LIN {X 0,Y 374.002,Z 352.596,A -85,B 0,C 180,E1 -14322.502,E2 -14322.502} C_VEL
LIN {X 0,Y 371.832,Z 350.324,A -85,B 0,C 180,E1 -14323.336,E2 -14323.336} C_VEL
LIN {X 0,Y 368.143,Z 347.333,A -85,B 0,C 180,E1 -14324.584,E2 -14324.584} C_VEL
LIN {X 0,Y 365.076,Z 343.836,A -85,B 0,C 180,E1 -14325.586,E2 -14325.586} C_VEL
LIN {X 0,Y 361.543,Z 340.851,A -85,B 0,C 180,E1 -14326.638,E2 -14326.638} C_VEL
LIN {X 0,Y 358.551,Z 337.452,A -85,B 0,C 180,E1 -14327.482,E2 -14327.482} C_VEL
LIN {X 0,Y 355.376,Z 334.461,A -85,B 0,C 180,E1 -14328.333,E2 -14328.333} C_VEL
LIN {X 0,Y 353.051,Z 331.524,A -85,B 0,C 180,E1 -14328.94,E2 -14328.94} C_VEL
LIN {X 0,Y 350.001,Z 328.379,A -85,B 0,C 180,E1 -14329.706,E2 -14329.706} C_VEL
LIN {X 0,Y 348.216,Z 325.956,A -85,B 0,C 180,E1 -14330.137,E2 -14330.137} C_VEL
LIN {X 0,Y 345.589,Z 323.181,A -85,B 0,C 180,E1 -14330.762,E2 -14330.762} C_VEL
LIN {X 0,Y 344.015,Z 320.684,A -85,B 0,C 180,E1 -14331.145,E2 -14331.145} C_VEL
LIN {X 0,Y 341.851,Z 318.515,A -85,B 0,C 180,E1 -14331.605,E2 -14331.605} C_VEL
LIN {X 0,Y 340.82,Z 316.079,A -85,B 0,C 180,E1 -14331.984,E2 -14331.984} C_VEL
LIN {X 0,Y 340.741,Z 315.556,A -85,B 0,C 180,E1 -14332.43,E2 -14332.43} C_VEL
LIN {X 0,Y 340.767,Z 315.54,A -85,B 0,C 180,E1 -14335.664,E2 -14335.664} C_VEL
LIN {X 0,Y 340.723,Z 315.529,A -85,B 0,C 180,E1 -14338.321,E2 -14338.321} C_VEL
LIN {X 0,Y 340.692,Z 315.544,A -85,B 0,C 180,E1 -14341.044,E2 -14341.044} C_VEL
LIN {X 0,Y 340.712,Z 315.516,A -85,B 0,C 180,E1 -14345.279,E2 -14345.279} C_VEL
LIN {X 0,Y 340.708,Z 315.545,A -85,B 0,C 180,E1 -14348.387,E2 -14348.387} C_VEL
LIN {X 0,Y 340.699,Z 315.5,A -85,B 0,C 180,E1 -14352.047,E2 -14352.047} C_VEL
LIN {X 0,Y 340.714,Z 315.539,A -85,B 0,C 180,E1 -14355.468,E2 -14355.468} C_VEL
LIN {X 0,Y 340.717,Z 315.533,A -85,B 0,C 180,E1 -14358.696,E2 -14358.696} C_VEL
LIN {X 0,Y 340.731,Z 315.543,A -85,B 0,C 180,E1 -14361.773,E2 -14361.773} C_VEL
LIN {X 0,Y 340.715,Z 315.527,A -85,B 0,C 180,E1 -14365.595,E2 -14365.595} C_VEL
LIN {X 0,Y 340.716,Z 315.541,A -85,B 0,C 180,E1 -14369.571,E2 -14369.571} C_VEL
LIN {X 0,Y 340.797,Z 315.511,A -85,B 0,C 180,E1 -14373.02,E2 -14373.02} C_VEL
LIN {X 0,Y 340.753,Z 315.53,A -85,B 0,C 180,E1 -14374.697,E2 -14374.697} C_VEL
LIN {X 0,Y 340.07,Z 315.623,A -85,B 0,C 180,E1 -14375.683,E2 -14375.683} C_VEL
LIN {X 0,Y 337.176,Z 315.983,A -85,B 0,C 180,E1 -14377.288,E2 -14377.288} C_VEL
LIN {X 0,Y 334.754,Z 316.278,A -85,B 0,C 180,E1 -14378.588,E2 -14378.588} C_VEL
LIN {X 0,Y 333.755,Z 316.39,A -85,B 0,C 180,E1 -14379.595,E2 -14379.595} C_VEL
LIN {X 0,Y 333.695,Z 316.393,A -85,B 0,C 180,E1 -14379.935,E2 -14379.935} C_VEL
LIN {X 0,Y 333.738,Z 316.399,A -85,B 0,C 180,E1 -14382.854,E2 -14382.854} C_VEL
LIN {X 0,Y 333.788,Z 316.405,A -85,B 0,C 180,E1 -14386.609,E2 -14386.609} C_VEL
LIN {X 0,Y 333.842,Z 316.365,A -85,B 0,C 180,E1 -14390.305,E2 -14390.305} C_VEL
LIN {X 0,Y 333.998,Z 316.371,A -85,B 0,C 180,E1 -14392.748,E2 -14392.748} C_VEL
LIN {X 0,Y 333.802,Z 316.404,A -85,B 0,C 180,E1 -14395.17,E2 -14395.17} C_VEL
LIN {X 0,Y 334.097,Z 316.353,A -85,B 0,C 180,E1 -14397.589,E2 -14397.589} C_VEL
LIN {X 0,Y 334.22,Z 316.316,A -85,B 0,C 180,E1 -14400.001,E2 -14400.001} C_VEL
LIN {X 0,Y 334.099,Z 316.357,A -85,B 0,C 180,E1 -14402.412,E2 -14402.412} C_VEL
LIN {X 0,Y 334.007,Z 316.377,A -85,B 0,C 180,E1 -14406.04,E2 -14406.04} C_VEL
LIN {X 0,Y 333.952,Z 316.357,A -85,B 0,C 180,E1 -14408.472,E2 -14408.472} C_VEL
LIN {X 0,Y 333.784,Z 316.395,A -85,B 0,C 180,E1 -14412.156,E2 -14412.156} C_VEL
LIN {X 0,Y 333.771,Z 316.402,A -85,B 0,C 180,E1 -14415.887,E2 -14415.887} C_VEL
LIN {X 0,Y 333.79,Z 316.376,A -85,B 0,C 180,E1 -14418.655,E2 -14418.655} C_VEL
LIN {X 0,Y 333.651,Z 316.421,A -85,B 0,C 180,E1 -14422.282,E2 -14422.282} C_VEL
LIN {X 0,Y 333.729,Z 316.391,A -85,B 0,C 180,E1 -14426.247,E2 -14426.247} C_VEL
LIN {X 0,Y 333.685,Z 316.415,A -85,B 0,C 180,E1 -14428.975,E2 -14428.975} C_VEL
LIN {X 0,Y 333.639,Z 316.414,A -85,B 0,C 180,E1 -14432.588,E2 -14432.588} C_VEL
LIN {X 0,Y 333.67,Z 316.417,A -85,B 0,C 180,E1 -14436.14,E2 -14436.14} C_VEL
LIN {X 0,Y 333.643,Z 316.416,A -85,B 0,C 180,E1 -14439.194,E2 -14439.194} C_VEL
LIN {X 0,Y 333.63,Z 316.427,A -85,B 0,C 180,E1 -14442.501,E2 -14442.501} C_VEL
LIN {X 0,Y 333.594,Z 316.432,A -85,B 0,C 180,E1 -14445.956,E2 -14445.956} C_VEL
LIN {X 0,Y 333.601,Z 316.404,A -85,B 0,C 180,E1 -14449.326,E2 -14449.326} C_VEL
LIN {X 0,Y 333.662,Z 316.414,A -85,B 0,C 180,E1 -14453.169,E2 -14453.169} C_VEL
LIN {X 0,Y 333.699,Z 316.565,A -85,B 0,C 180,E1 -14456.885,E2 -14456.885} C_VEL
LIN {X 0,Y 335.008,Z 322.928,A -85,B 0,C 180,E1 -14459.332,E2 -14459.332} C_VEL
LIN {X 0,Y 336.868,Z 332.516,A -85,B 0,C 180,E1 -14462.679,E2 -14462.679} C_VEL
LIN {X 0,Y 337.066,Z 336.458,A -85,B 0,C 180,E1 -14464.033,E2 -14464.033} C_VEL
LIN {X 0,Y 336.29,Z 342.314,A -85,B 0,C 180,E1 -14465.915,E2 -14465.915} C_VEL
LIN {X 0,Y 336.975,Z 345.953,A -85,B 0,C 180,E1 -14466.117,E2 -14466.117} C_VEL
LIN {X 0,Y 342.072,Z 371.242,A -85,B 0,C 180,E1 -14467.057,E2 -14467.057} C_VEL
LIN {X 0,Y 343.729,Z 381.109,A -85,B 0,C 180,E1 -14467.391,E2 -14467.391} C_VEL
LIN {X 0,Y 342.454,Z 447.28,A -85,B 0,C 180,E1 -14468.795,E2 -14468.795} C_VEL
LIN {X 0,Y 341.879,Z 458.022,A -85,B 0,C 180,E1 -14469.152,E2 -14469.152} C_VEL
LIN {X 0,Y 341.242,Z 467.12,A -85,B 0,C 180,E1 -14469.585,E2 -14469.585} C_VEL
LIN {X 0,Y 340.44,Z 476.473,A -85,B 0,C 180,E1 -14470.164,E2 -14470.164} C_VEL
LIN {X 0,Y 339.419,Z 486.611,A -85,B 0,C 180,E1 -14470.967,E2 -14470.967} C_VEL
LIN {X 0,Y 338.379,Z 495.605,A -85,B 0,C 180,E1 -14471.848,E2 -14471.848} C_VEL
LIN {X 0,Y 337.286,Z 504.331,A -85,B 0,C 180,E1 -14472.884,E2 -14472.884} C_VEL
LIN {X 0,Y 336.298,Z 512.266,A -85,B 0,C 180,E1 -14474.013,E2 -14474.013} C_VEL
LIN {X 0,Y 335.469,Z 518.947,A -85,B 0,C 180,E1 -14475.13,E2 -14475.13} C_VEL
LIN {X 0,Y 334.69,Z 525.15,A -85,B 0,C 180,E1 -14476.336,E2 -14476.336} C_VEL
LIN {X 0,Y 333.743,Z 531.685,A -85,B 0,C 180,E1 -14477.844,E2 -14477.844} C_VEL
LIN {X 0,Y 333.24,Z 536.189,A -85,B 0,C 180,E1 -14479.059,E2 -14479.059} C_VEL
LIN {X 0,Y 332.611,Z 541.681,A -85,B 0,C 180,E1 -14480.882,E2 -14480.882} C_VEL
LIN {X 0,Y 332.203,Z 546.006,A -85,B 0,C 180,E1 -14482.708,E2 -14482.708} C_VEL
LIN {X 0,Y 332.034,Z 548.743,A -85,B 0,C 180,E1 -14484.174,E2 -14484.174} C_VEL
LIN {X 0,Y 331.97,Z 551.563,A -85,B 0,C 180,E1 -14486.359,E2 -14486.359} C_VEL
LIN {X 0,Y 331.916,Z 552.621,A -85,B 0,C 180,E1 -14487.573,E2 -14487.573} C_VEL
LIN {X 0,Y 331.913,Z 553.21,A -85,B 0,C 180,E1 -14488.787,E2 -14488.787} C_VEL
LIN {X 0,Y 331.913,Z 553.21,A -85,B 0,C 180,E1 -14491.213,E2 -14491.213} C_VEL
LIN {X 0,Y 331.916,Z 552.621,A -85,B 0,C 180,E1 -14492.427,E2 -14492.427} C_VEL
LIN {X 0,Y 331.971,Z 550.174,A -85,B 0,C 180,E1 -14494.858,E2 -14494.858} C_VEL
LIN {X 0,Y 332.106,Z 547.223,A -85,B 0,C 180,E1 -14496.684,E2 -14496.684} C_VEL
LIN {X 0,Y 332.467,Z 543.235,A -85,B 0,C 180,E1 -14498.509,E2 -14498.509} C_VEL
LIN {X 0,Y 332.988,Z 538.104,A -85,B 0,C 180,E1 -14500.335,E2 -14500.335} C_VEL
LIN {X 0,Y 333.597,Z 532.841,A -85,B 0,C 180,E1 -14501.853,E2 -14501.853} C_VEL
LIN {X 0,Y 334.485,Z 526.526,A -85,B 0,C 180,E1 -14503.363,E2 -14503.363} C_VEL
LIN {X 0,Y 335.255,Z 520.574,A -85,B 0,C 180,E1 -14504.569,E2 -14504.569} C_VEL
LIN {X 0,Y 336.287,Z 512.309,A -85,B 0,C 180,E1 -14505.981,E2 -14505.981} C_VEL
LIN {X 0,Y 337.288,Z 504.331,A -85,B 0,C 180,E1 -14507.116,E2 -14507.116} C_VEL
LIN {X 0,Y 338.395,Z 495.606,A -85,B 0,C 180,E1 -14508.151,E2 -14508.151} C_VEL
LIN {X 0,Y 339.445,Z 486.612,A -85,B 0,C 180,E1 -14509.031,E2 -14509.031} C_VEL
LIN {X 0,Y 340.43,Z 476.472,A -85,B 0,C 180,E1 -14509.836,E2 -14509.836} C_VEL
LIN {X 0,Y 341.444,Z 464.545,A -85,B 0,C 180,E1 -14510.56,E2 -14510.56} C_VEL
LIN {X 0,Y 342.275,Z 451.253,A -85,B 0,C 180,E1 -14511.098,E2 -14511.098} C_VEL
LIN {X 0,Y 342.789,Z 432.475,A -85,B 0,C 180,E1 -14511.538,E2 -14511.538} C_VEL
LIN {X 0,Y 343.621,Z 380.01,A -85,B 0,C 180,E1 -14512.641,E2 -14512.641} C_VEL
LIN {X 0,Y 338.297,Z 352.082,A -85,B 0,C 180,E1 -14513.646,E2 -14513.646} C_VEL
LIN {X 0,Y 336.284,Z 342.655,A -85,B 0,C 180,E1 -14514.04,E2 -14514.04} C_VEL
LIN {X 0,Y 336.385,Z 341.162,A -85,B 0,C 180,E1 -14514.402,E2 -14514.402} C_VEL
LIN {X 0,Y 337.123,Z 335.439,A -85,B 0,C 180,E1 -14516.307,E2 -14516.307} C_VEL
LIN {X 0,Y 336.548,Z 330.722,A -85,B 0,C 180,E1 -14517.961,E2 -14517.961} C_VEL
LIN {X 0,Y 334.829,Z 322.015,A -85,B 0,C 180,E1 -14521.09,E2 -14521.09} C_VEL
LIN {X 0,Y 333.672,Z 316.471,A -85,B 0,C 180,E1 -14523.203,E2 -14523.203} C_VEL
LIN {X 0,Y 333.662,Z 316.414,A -85,B 0,C 180,E1 -14526.831,E2 -14526.831} C_VEL
LIN {X 0,Y 333.602,Z 316.404,A -85,B 0,C 180,E1 -14530.773,E2 -14530.773} C_VEL
LIN {X 0,Y 333.591,Z 316.43,A -85,B 0,C 180,E1 -14534.249,E2 -14534.249} C_VEL
LIN {X 0,Y 333.639,Z 316.427,A -85,B 0,C 180,E1 -14537.617,E2 -14537.617} C_VEL
LIN {X 0,Y 333.649,Z 316.416,A -85,B 0,C 180,E1 -14541.201,E2 -14541.201} C_VEL
LIN {X 0,Y 333.67,Z 316.417,A -85,B 0,C 180,E1 -14543.86,E2 -14543.86} C_VEL
LIN {X 0,Y 333.639,Z 316.414,A -85,B 0,C 180,E1 -14547.412,E2 -14547.412} C_VEL
LIN {X 0,Y 333.685,Z 316.415,A -85,B 0,C 180,E1 -14551.025,E2 -14551.025} C_VEL
LIN {X 0,Y 333.729,Z 316.391,A -85,B 0,C 180,E1 -14553.753,E2 -14553.753} C_VEL
LIN {X 0,Y 333.651,Z 316.421,A -85,B 0,C 180,E1 -14557.718,E2 -14557.718} C_VEL
LIN {X 0,Y 333.787,Z 316.377,A -85,B 0,C 180,E1 -14561.588,E2 -14561.588} C_VEL
LIN {X 0,Y 333.802,Z 316.405,A -85,B 0,C 180,E1 -14565.576,E2 -14565.576} C_VEL
LIN {X 0,Y 333.827,Z 316.377,A -85,B 0,C 180,E1 -14569.077,E2 -14569.077} C_VEL
LIN {X 0,Y 333.999,Z 316.366,A -85,B 0,C 180,E1 -14572.746,E2 -14572.746} C_VEL
LIN {X 0,Y 333.802,Z 316.406,A -85,B 0,C 180,E1 -14575.168,E2 -14575.168} C_VEL
LIN {X 0,Y 334.099,Z 316.357,A -85,B 0,C 180,E1 -14577.588,E2 -14577.588} C_VEL
LIN {X 0,Y 334.22,Z 316.316,A -85,B 0,C 180,E1 -14579.999,E2 -14579.999} C_VEL
LIN {X 0,Y 334.097,Z 316.353,A -85,B 0,C 180,E1 -14582.411,E2 -14582.411} C_VEL
LIN {X 0,Y 333.983,Z 316.373,A -85,B 0,C 180,E1 -14586.674,E2 -14586.674} C_VEL
LIN {X 0,Y 333.842,Z 316.365,A -85,B 0,C 180,E1 -14589.695,E2 -14589.695} C_VEL
LIN {X 0,Y 333.788,Z 316.405,A -85,B 0,C 180,E1 -14593.391,E2 -14593.391} C_VEL
LIN {X 0,Y 333.738,Z 316.399,A -85,B 0,C 180,E1 -14597.146,E2 -14597.146} C_VEL
LIN {X 0,Y 333.729,Z 316.388,A -85,B 0,C 180,E1 -14599.69,E2 -14599.69} C_VEL
LIN {X 0,Y 333.684,Z 316.415,A -85,B 0,C 180,E1 -14602.278,E2 -14602.278} C_VEL
LIN {X 0,Y 333.728,Z 316.398,A -85,B 0,C 180,E1 -14606.246,E2 -14606.246} C_VEL
LIN {X 0,Y 333.703,Z 316.404,A -85,B 0,C 180,E1 -14608.972,E2 -14608.972} C_VEL
LIN {X 0,Y 333.638,Z 316.421,A -85,B 0,C 180,E1 -14612.588,E2 -14612.588} C_VEL
LIN {X 0,Y 333.669,Z 316.414,A -85,B 0,C 180,E1 -14616.139,E2 -14616.139} C_VEL
LIN {X 0,Y 333.677,Z 316.415,A -85,B 0,C 180,E1 -14619.187,E2 -14619.187} C_VEL
LIN {X 0,Y 333.681,Z 316.417,A -85,B 0,C 180,E1 -14622.511,E2 -14622.511} C_VEL
LIN {X 0,Y 333.628,Z 316.401,A -85,B 0,C 180,E1 -14625.962,E2 -14625.962} C_VEL
LIN {X 0,Y 333.648,Z 316.388,A -85,B 0,C 180,E1 -14629.314,E2 -14629.314} C_VEL
LIN {X 0,Y 333.649,Z 316.427,A -85,B 0,C 180,E1 -14632.35,E2 -14632.35} C_VEL
LIN {X 0,Y 333.668,Z 316.39,A -85,B 0,C 180,E1 -14635.342,E2 -14635.342} C_VEL
LIN {X 0,Y 333.684,Z 316.406,A -85,B 0,C 180,E1 -14639.637,E2 -14639.637} C_VEL
LIN {X 0,Y 333.734,Z 316.411,A -85,B 0,C 180,E1 -14642.401,E2 -14642.401} C_VEL
LIN {X 0,Y 333.722,Z 316.418,A -85,B 0,C 180,E1 -14645.091,E2 -14645.091} C_VEL
LIN {X 0,Y 333.713,Z 316.564,A -85,B 0,C 180,E1 -14646.636,E2 -14646.636} C_VEL
LIN {X 0,Y 333.901,Z 317.484,A -85,B 0,C 180,E1 -14646.906,E2 -14646.906} C_VEL
LIN {X 0,Y 335.44,Z 320.272,A -85,B 0,C 180,E1 -14647.294,E2 -14647.294} C_VEL
LIN {X 0,Y 337.24,Z 322.145,A -85,B 0,C 180,E1 -14647.649,E2 -14647.649} C_VEL
LIN {X 0,Y 339.606,Z 325.545,A -85,B 0,C 180,E1 -14648.193,E2 -14648.193} C_VEL
LIN {X 0,Y 341.243,Z 327.304,A -85,B 0,C 180,E1 -14648.55,E2 -14648.55} C_VEL
LIN {X 0,Y 344.017,Z 330.834,A -85,B 0,C 180,E1 -14649.167,E2 -14649.167} C_VEL
LIN {X 0,Y 346.131,Z 333.088,A -85,B 0,C 180,E1 -14649.669,E2 -14649.669} C_VEL
LIN {X 0,Y 349.257,Z 336.713,A -85,B 0,C 180,E1 -14650.409,E2 -14650.409} C_VEL
LIN {X 0,Y 351.305,Z 338.801,A -85,B 0,C 180,E1 -14650.915,E2 -14650.915} C_VEL
LIN {X 0,Y 354.984,Z 342.849,A -85,B 0,C 180,E1 -14651.859,E2 -14651.859} C_VEL
LIN {X 0,Y 357.12,Z 344.835,A -85,B 0,C 180,E1 -14652.431,E2 -14652.431} C_VEL
LIN {X 0,Y 360.924,Z 348.801,A -85,B 0,C 180,E1 -14653.498,E2 -14653.498} C_VEL
LIN {X 0,Y 363.731,Z 351.163,A -85,B 0,C 180,E1 -14654.333,E2 -14654.333} C_VEL
LIN {X 0,Y 367.168,Z 354.797,A -85,B 0,C 180,E1 -14655.432,E2 -14655.432} C_VEL
LIN {X 0,Y 371.068,Z 357.902,A -85,B 0,C 180,E1 -14656.751,E2 -14656.751} C_VEL
LIN {X 0,Y 374.707,Z 361.571,A -85,B 0,C 180,E1 -14658.165,E2 -14658.165} C_VEL
LIN {X 0,Y 378.245,Z 364.068,A -85,B 0,C 180,E1 -14659.673,E2 -14659.673} C_VEL
LIN {X 0,Y 379.884,Z 365.154,A -85,B 0,C 180,E1 -14660.464,E2 -14660.464} C_VEL
LIN {X 0,Y 382.521,Z 368.124,A -85,B 0,C 180,E1 -14661.961,E2 -14661.961} C_VEL
LIN {X 0,Y 384.968,Z 370.062,A -85,B 0,C 180,E1 -14663.58,E2 -14663.58} C_VEL
LIN {X 0,Y 387.283,Z 371.337,A -85,B 0,C 180,E1 -14665.578,E2 -14665.578} C_VEL
LIN {X 0,Y 388.664,Z 371.823,A -85,B 0,C 180,E1 -14667.428,E2 -14667.428} C_VEL
LIN {X 0,Y 389.239,Z 372.261,A -85,B 0,C 180,E1 -14668.965,E2 -14668.965} C_VEL
LIN {X 0,Y 389.407,Z 372.18,A -85,B 0,C 180,E1 -14670,E2 -14670} C_VEL
LIN {X 0,Y 389.126,Z 372.136,A -85,B 0,C 180,E1 -14671.552,E2 -14671.552} C_VEL
LIN {X 0,Y 388.36,Z 371.702,A -85,B 0,C 180,E1 -14673.112,E2 -14673.112} C_VEL
LIN {X 0,Y 386.736,Z 371.099,A -85,B 0,C 180,E1 -14674.943,E2 -14674.943} C_VEL
LIN {X 0,Y 384.56,Z 369.785,A -85,B 0,C 180,E1 -14676.7,E2 -14676.7} C_VEL
LIN {X 0,Y 382.058,Z 367.692,A -85,B 0,C 180,E1 -14678.309,E2 -14678.309} C_VEL
LIN {X 0,Y 379.212,Z 364.566,A -85,B 0,C 180,E1 -14679.865,E2 -14679.865} C_VEL
LIN {X 0,Y 375.944,Z 362.622,A -85,B 0,C 180,E1 -14681.307,E2 -14681.307} C_VEL
LIN {X 0,Y 372.666,Z 359.673,A -85,B 0,C 180,E1 -14682.629,E2 -14682.629} C_VEL
LIN {X 0,Y 370.003,Z 356.954,A -85,B 0,C 180,E1 -14683.635,E2 -14683.635} C_VEL
LIN {X 0,Y 365.937,Z 353.626,A -85,B 0,C 180,E1 -14684.976,E2 -14684.976} C_VEL
LIN {X 0,Y 362.653,Z 350.169,A -85,B 0,C 180,E1 -14685.995,E2 -14685.995} C_VEL
LIN {X 0,Y 358.82,Z 346.809,A -85,B 0,C 180,E1 -14687.085,E2 -14687.085} C_VEL
LIN {X 0,Y 355.812,Z 343.521,A -85,B 0,C 180,E1 -14687.928,E2 -14687.928} C_VEL
LIN {X 0,Y 352.062,Z 339.815,A -85,B 0,C 180,E1 -14688.881,E2 -14688.881} C_VEL
LIN {X 0,Y 350.013,Z 337.385,A -85,B 0,C 180,E1 -14689.415,E2 -14689.415} C_VEL
LIN {X 0,Y 346.537,Z 333.696,A -85,B 0,C 180,E1 -14690.229,E2 -14690.229} C_VEL
LIN {X 0,Y 344.964,Z 331.748,A -85,B 0,C 180,E1 -14690.614,E2 -14690.614} C_VEL
LIN {X 0,Y 341.952,Z 328.424,A -85,B 0,C 180,E1 -14691.286,E2 -14691.286} C_VEL
LIN {X 0,Y 340.285,Z 326.164,A -85,B 0,C 180,E1 -14691.661,E2 -14691.661} C_VEL
LIN {X 0,Y 337.899,Z 323.317,A -85,B 0,C 180,E1 -14692.197,E2 -14692.197} C_VEL
LIN {X 0,Y 336.543,Z 321.282,A -85,B 0,C 180,E1 -14692.493,E2 -14692.493} C_VEL
LIN {X 0,Y 334.616,Z 319.146,A -85,B 0,C 180,E1 -14692.878,E2 -14692.878} C_VEL
LIN {X 0,Y 333.801,Z 317.073,A -85,B 0,C 180,E1 -14693.17,E2 -14693.17} C_VEL
LIN {X 0,Y 333.679,Z 316.494,A -85,B 0,C 180,E1 -14693.425,E2 -14693.425} C_VEL
LIN {X 0,Y 333.73,Z 316.416,A -85,B 0,C 180,E1 -14696.246,E2 -14696.246} C_VEL
LIN {X 0,Y 333.684,Z 316.4,A -85,B 0,C 180,E1 -14698.974,E2 -14698.974} C_VEL
LIN {X 0,Y 333.637,Z 316.42,A -85,B 0,C 180,E1 -14702.587,E2 -14702.587} C_VEL
LIN {X 0,Y 333.671,Z 316.404,A -85,B 0,C 180,E1 -14706.139,E2 -14706.139} C_VEL
LIN {X 0,Y 333.664,Z 316.414,A -85,B 0,C 180,E1 -14709.189,E2 -14709.189} C_VEL
LIN {X 0,Y 333.631,Z 316.38,A -85,B 0,C 180,E1 -14712.501,E2 -14712.501} C_VEL
LIN {X 0,Y 333.661,Z 316.423,A -85,B 0,C 180,E1 -14715.967,E2 -14715.967} C_VEL
LIN {X 0,Y 333.694,Z 316.405,A -85,B 0,C 180,E1 -14719.304,E2 -14719.304} C_VEL
LIN {X 0,Y 333.658,Z 316.422,A -85,B 0,C 180,E1 -14723.168,E2 -14723.168} C_VEL
LIN {X 0,Y 333.631,Z 316.415,A -85,B 0,C 180,E1 -14726.792,E2 -14726.792} C_VEL
LIN {X 0,Y 333.695,Z 316.416,A -85,B 0,C 180,E1 -14729.71,E2 -14729.71} C_VEL
LIN {X 0,Y 333.736,Z 316.39,A -85,B 0,C 180,E1 -14732.401,E2 -14732.401} C_VEL
LIN {X 0,Y 333.718,Z 316.41,A -85,B 0,C 180,E1 -14735.091,E2 -14735.091} C_VEL
LIN {X 0,Y 333.672,Z 316.406,A -85,B 0,C 180,E1 -14739.019,E2 -14739.019} C_VEL
LIN {X 0,Y 333.695,Z 316.393,A -85,B 0,C 180,E1 -14739.935,E2 -14739.935} C_VEL
LIN {X 0,Y 333.085,Z 316.469,A -85,B 0,C 180,E1 -14740.943,E2 -14740.943} C_VEL
LIN {X 0,Y 330.261,Z 316.836,A -85,B 0,C 180,E1 -14742.582,E2 -14742.582} C_VEL
LIN {X 0,Y 327.845,Z 317.148,A -85,B 0,C 180,E1 -14743.91,E2 -14743.91} C_VEL
LIN {X 0,Y 326.823,Z 317.277,A -85,B 0,C 180,E1 -14744.938,E2 -14744.938} C_VEL
LIN {X 0,Y 326.75,Z 317.284,A -85,B 0,C 180,E1 -14745.286,E2 -14745.286} C_VEL
LIN {X 0,Y 326.761,Z 317.253,A -85,B 0,C 180,E1 -14748.839,E2 -14748.839} C_VEL
LIN {X 0,Y 326.95,Z 317.247,A -85,B 0,C 180,E1 -14752.59,E2 -14752.59} C_VEL
LIN {X 0,Y 326.768,Z 317.281,A -85,B 0,C 180,E1 -14755.065,E2 -14755.065} C_VEL
LIN {X 0,Y 327.038,Z 317.232,A -85,B 0,C 180,E1 -14757.537,E2 -14757.537} C_VEL
LIN {X 0,Y 327.172,Z 317.193,A -85,B 0,C 180,E1 -14760.001,E2 -14760.001} C_VEL
LIN {X 0,Y 327.04,Z 317.236,A -85,B 0,C 180,E1 -14762.464,E2 -14762.464} C_VEL
LIN {X 0,Y 326.982,Z 317.252,A -85,B 0,C 180,E1 -14766.17,E2 -14766.17} C_VEL
LIN {X 0,Y 326.799,Z 317.241,A -85,B 0,C 180,E1 -14769.907,E2 -14769.907} C_VEL
LIN {X 0,Y 326.753,Z 317.279,A -85,B 0,C 180,E1 -14773.686,E2 -14773.686} C_VEL
LIN {X 0,Y 326.693,Z 317.266,A -85,B 0,C 180,E1 -14777.529,E2 -14777.529} C_VEL
LIN {X 0,Y 326.652,Z 317.275,A -85,B 0,C 180,E1 -14780.136,E2 -14780.136} C_VEL
LIN {X 0,Y 326.643,Z 317.293,A -85,B 0,C 180,E1 -14784.13,E2 -14784.13} C_VEL
LIN {X 0,Y 326.678,Z 317.267,A -85,B 0,C 180,E1 -14786.859,E2 -14786.859} C_VEL
LIN {X 0,Y 326.63,Z 317.299,A -85,B 0,C 180,E1 -14790.611,E2 -14790.611} C_VEL
LIN {X 0,Y 326.602,Z 317.282,A -85,B 0,C 180,E1 -14794.021,E2 -14794.021} C_VEL
LIN {X 0,Y 326.623,Z 317.298,A -85,B 0,C 180,E1 -14797.239,E2 -14797.239} C_VEL
LIN {X 0,Y 326.575,Z 317.301,A -85,B 0,C 180,E1 -14801.132,E2 -14801.132} C_VEL
LIN {X 0,Y 326.525,Z 317.305,A -85,B 0,C 180,E1 -14804.744,E2 -14804.744} C_VEL
LIN {X 0,Y 326.561,Z 317.29,A -85,B 0,C 180,E1 -14808.153,E2 -14808.153} C_VEL
LIN {X 0,Y 326.581,Z 317.301,A -85,B 0,C 180,E1 -14811.387,E2 -14811.387} C_VEL
LIN {X 0,Y 326.618,Z 317.286,A -85,B 0,C 180,E1 -14814.853,E2 -14814.853} C_VEL
LIN {X 0,Y 326.672,Z 317.479,A -85,B 0,C 180,E1 -14816.487,E2 -14816.487} C_VEL
LIN {X 0,Y 328.006,Z 324.056,A -85,B 0,C 180,E1 -14819.055,E2 -14819.055} C_VEL
LIN {X 0,Y 329.631,Z 332.307,A -85,B 0,C 180,E1 -14822.028,E2 -14822.028} C_VEL
LIN {X 0,Y 330.177,Z 336.26,A -85,B 0,C 180,E1 -14823.45,E2 -14823.45} C_VEL
LIN {X 0,Y 329.446,Z 342.132,A -85,B 0,C 180,E1 -14825.385,E2 -14825.385} C_VEL
LIN {X 0,Y 330.305,Z 346.413,A -85,B 0,C 180,E1 -14825.619,E2 -14825.619} C_VEL
LIN {X 0,Y 335.111,Z 370.101,A -85,B 0,C 180,E1 -14826.53,E2 -14826.53} C_VEL
LIN {X 0,Y 337.185,Z 382.571,A -85,B 0,C 180,E1 -14826.965,E2 -14826.965} C_VEL
LIN {X 0,Y 335.845,Z 447.093,A -85,B 0,C 180,E1 -14828.357,E2 -14828.357} C_VEL
LIN {X 0,Y 335.267,Z 457.829,A -85,B 0,C 180,E1 -14828.721,E2 -14828.721} C_VEL
LIN {X 0,Y 334.61,Z 466.926,A -85,B 0,C 180,E1 -14829.161,E2 -14829.161} C_VEL
LIN {X 0,Y 333.75,Z 476.278,A -85,B 0,C 180,E1 -14829.749,E2 -14829.749} C_VEL
LIN {X 0,Y 332.695,Z 486.417,A -85,B 0,C 180,E1 -14830.567,E2 -14830.567} C_VEL
LIN {X 0,Y 331.616,Z 495.411,A -85,B 0,C 180,E1 -14831.465,E2 -14831.465} C_VEL
LIN {X 0,Y 330.49,Z 504.137,A -85,B 0,C 180,E1 -14832.52,E2 -14832.52} C_VEL
LIN {X 0,Y 329.478,Z 511.897,A -85,B 0,C 180,E1 -14833.644,E2 -14833.644} C_VEL
LIN {X 0,Y 328.582,Z 518.809,A -85,B 0,C 180,E1 -14834.822,E2 -14834.822} C_VEL
LIN {X 0,Y 327.778,Z 524.956,A -85,B 0,C 180,E1 -14836.042,E2 -14836.042} C_VEL
LIN {X 0,Y 326.779,Z 531.49,A -85,B 0,C 180,E1 -14837.581,E2 -14837.581} C_VEL
LIN {X 0,Y 326.216,Z 535.993,A -85,B 0,C 180,E1 -14838.82,E2 -14838.82} C_VEL
LIN {X 0,Y 325.578,Z 541.486,A -85,B 0,C 180,E1 -14840.683,E2 -14840.683} C_VEL
LIN {X 0,Y 325.154,Z 545.812,A -85,B 0,C 180,E1 -14842.549,E2 -14842.549} C_VEL
LIN {X 0,Y 324.926,Z 548.844,A -85,B 0,C 180,E1 -14844.251,E2 -14844.251} C_VEL
LIN {X 0,Y 324.877,Z 551.369,A -85,B 0,C 180,E1 -14846.279,E2 -14846.279} C_VEL
LIN {X 0,Y 324.835,Z 552.427,A -85,B 0,C 180,E1 -14847.52,E2 -14847.52} C_VEL
LIN {X 0,Y 324.822,Z 553.016,A -85,B 0,C 180,E1 -14848.76,E2 -14848.76} C_VEL
LIN {X 0,Y 324.822,Z 553.016,A -85,B 0,C 180,E1 -14851.24,E2 -14851.24} C_VEL
LIN {X 0,Y 324.835,Z 552.427,A -85,B 0,C 180,E1 -14852.48,E2 -14852.48} C_VEL
LIN {X 0,Y 324.882,Z 549.979,A -85,B 0,C 180,E1 -14854.964,E2 -14854.964} C_VEL
LIN {X 0,Y 325.047,Z 547.029,A -85,B 0,C 180,E1 -14856.83,E2 -14856.83} C_VEL
LIN {X 0,Y 325.406,Z 543.04,A -85,B 0,C 180,E1 -14858.695,E2 -14858.695} C_VEL
LIN {X 0,Y 325.968,Z 537.909,A -85,B 0,C 180,E1 -14860.56,E2 -14860.56} C_VEL
LIN {X 0,Y 326.628,Z 532.646,A -85,B 0,C 180,E1 -14862.11,E2 -14862.11} C_VEL
LIN {X 0,Y 327.57,Z 526.331,A -85,B 0,C 180,E1 -14863.651,E2 -14863.651} C_VEL
LIN {X 0,Y 328.346,Z 520.379,A -85,B 0,C 180,E1 -14864.883,E2 -14864.883} C_VEL
LIN {X 0,Y 329.338,Z 512.888,A -85,B 0,C 180,E1 -14866.199,E2 -14866.199} C_VEL
LIN {X 0,Y 330.332,Z 505.271,A -85,B 0,C 180,E1 -14867.329,E2 -14867.329} C_VEL
LIN {X 0,Y 331.498,Z 496.764,A -85,B 0,C 180,E1 -14868.382,E2 -14868.382} C_VEL
LIN {X 0,Y 332.563,Z 488.05,A -85,B 0,C 180,E1 -14869.28,E2 -14869.28} C_VEL
LIN {X 0,Y 333.576,Z 478.293,A -85,B 0,C 180,E1 -14870.101,E2 -14870.101} C_VEL
LIN {X 0,Y 334.398,Z 469.501,A -85,B 0,C 180,E1 -14870.692,E2 -14870.692} C_VEL
LIN {X 0,Y 335.115,Z 459.576,A -85,B 0,C 180,E1 -14871.208,E2 -14871.208} C_VEL
LIN {X 0,Y 335.735,Z 449.728,A -85,B 0,C 180,E1 -14871.57,E2 -14871.57} C_VEL
LIN {X 0,Y 336.287,Z 428.702,A -85,B 0,C 180,E1 -14872.056,E2 -14872.056} C_VEL
LIN {X 0,Y 337.081,Z 381.176,A -85,B 0,C 180,E1 -14873.075,E2 -14873.075} C_VEL
LIN {X 0,Y 332.125,Z 354.829,A -85,B 0,C 180,E1 -14874.045,E2 -14874.045} C_VEL
LIN {X 0,Y 329.474,Z 342.433,A -85,B 0,C 180,E1 -14874.572,E2 -14874.572} C_VEL
LIN {X 0,Y 329.57,Z 340.965,A -85,B 0,C 180,E1 -14874.941,E2 -14874.941} C_VEL
LIN {X 0,Y 330.155,Z 336.089,A -85,B 0,C 180,E1 -14876.612,E2 -14876.612} C_VEL
LIN {X 0,Y 329.18,Z 329.742,A -85,B 0,C 180,E1 -14878.912,E2 -14878.912} C_VEL
LIN {X 0,Y 327.232,Z 320.188,A -85,B 0,C 180,E1 -14882.474,E2 -14882.474} C_VEL
LIN {X 0,Y 326.639,Z 317.378,A -85,B 0,C 180,E1 -14883.587,E2 -14883.587} C_VEL
LIN {X 0,Y 326.622,Z 317.296,A -85,B 0,C 180,E1 -14887.236,E2 -14887.236} C_VEL
LIN {X 0,Y 326.542,Z 317.285,A -85,B 0,C 180,E1 -14891.123,E2 -14891.123} C_VEL
LIN {X 0,Y 326.559,Z 317.309,A -85,B 0,C 180,E1 -14893.525,E2 -14893.525} C_VEL
LIN {X 0,Y 326.574,Z 317.303,A -85,B 0,C 180,E1 -14897.027,E2 -14897.027} C_VEL
LIN {X 0,Y 326.608,Z 317.292,A -85,B 0,C 180,E1 -14900.772,E2 -14900.772} C_VEL
LIN {X 0,Y 326.607,Z 317.292,A -85,B 0,C 180,E1 -14904.479,E2 -14904.479} C_VEL
LIN {X 0,Y 326.604,Z 317.29,A -85,B 0,C 180,E1 -14907.454,E2 -14907.454} C_VEL
LIN {X 0,Y 326.643,Z 317.293,A -85,B 0,C 180,E1 -14910.339,E2 -14910.339} C_VEL
LIN {X 0,Y 326.685,Z 317.276,A -85,B 0,C 180,E1 -14914.515,E2 -14914.515} C_VEL
LIN {X 0,Y 326.614,Z 317.294,A -85,B 0,C 180,E1 -14918.542,E2 -14918.542} C_VEL
LIN {X 0,Y 326.739,Z 317.254,A -85,B 0,C 180,E1 -14921.177,E2 -14921.177} C_VEL
LIN {X 0,Y 326.757,Z 317.281,A -85,B 0,C 180,E1 -14925.432,E2 -14925.432} C_VEL
LIN {X 0,Y 326.763,Z 317.26,A -85,B 0,C 180,E1 -14928.838,E2 -14928.838} C_VEL
LIN {X 0,Y 326.951,Z 317.243,A -85,B 0,C 180,E1 -14932.589,E2 -14932.589} C_VEL
LIN {X 0,Y 326.769,Z 317.281,A -85,B 0,C 180,E1 -14935.064,E2 -14935.064} C_VEL
LIN {X 0,Y 327.04,Z 317.236,A -85,B 0,C 180,E1 -14937.536,E2 -14937.536} C_VEL
LIN {X 0,Y 327.172,Z 317.193,A -85,B 0,C 180,E1 -14939.999,E2 -14939.999} C_VEL
LIN {X 0,Y 327.038,Z 317.232,A -85,B 0,C 180,E1 -14942.463,E2 -14942.463} C_VEL
LIN {X 0,Y 326.95,Z 317.25,A -85,B 0,C 180,E1 -14946.666,E2 -14946.666} C_VEL
LIN {X 0,Y 326.797,Z 317.241,A -85,B 0,C 180,E1 -14949.906,E2 -14949.906} C_VEL
LIN {X 0,Y 326.751,Z 317.282,A -85,B 0,C 180,E1 -14953.685,E2 -14953.685} C_VEL
LIN {X 0,Y 326.691,Z 317.273,A -85,B 0,C 180,E1 -14957.528,E2 -14957.528} C_VEL
LIN {X 0,Y 326.655,Z 317.272,A -85,B 0,C 180,E1 -14960.135,E2 -14960.135} C_VEL
LIN {X 0,Y 326.644,Z 317.295,A -85,B 0,C 180,E1 -14964.129,E2 -14964.129} C_VEL
LIN {X 0,Y 326.677,Z 317.27,A -85,B 0,C 180,E1 -14966.857,E2 -14966.857} C_VEL
LIN {X 0,Y 326.631,Z 317.298,A -85,B 0,C 180,E1 -14970.611,E2 -14970.611} C_VEL
LIN {X 0,Y 326.6,Z 317.286,A -85,B 0,C 180,E1 -14974.019,E2 -14974.019} C_VEL
LIN {X 0,Y 326.622,Z 317.301,A -85,B 0,C 180,E1 -14977.239,E2 -14977.239} C_VEL
LIN {X 0,Y 326.628,Z 317.286,A -85,B 0,C 180,E1 -14980.203,E2 -14980.203} C_VEL
LIN {X 0,Y 326.611,Z 317.3,A -85,B 0,C 180,E1 -14983.516,E2 -14983.516} C_VEL
LIN {X 0,Y 326.582,Z 317.261,A -85,B 0,C 180,E1 -14987.026,E2 -14987.026} C_VEL
LIN {X 0,Y 326.626,Z 317.29,A -85,B 0,C 180,E1 -14990.768,E2 -14990.768} C_VEL
LIN {X 0,Y 326.607,Z 317.274,A -85,B 0,C 180,E1 -14994.481,E2 -14994.481} C_VEL
LIN {X 0,Y 326.602,Z 317.296,A -85,B 0,C 180,E1 -14997.456,E2 -14997.456} C_VEL
LIN {X 0,Y 326.642,Z 317.277,A -85,B 0,C 180,E1 -15000.34,E2 -15000.34} C_VEL
LIN {X 0,Y 326.685,Z 317.294,A -85,B 0,C 180,E1 -15004.516,E2 -15004.516} C_VEL
LIN {X 0,Y 326.69,Z 317.588,A -85,B 0,C 180,E1 -15005.621,E2 -15005.621} C_VEL
LIN {X 0,Y 327.047,Z 318.932,A -85,B 0,C 180,E1 -15005.866,E2 -15005.866} C_VEL
LIN {X 0,Y 328.752,Z 321.563,A -85,B 0,C 180,E1 -15006.21,E2 -15006.21} C_VEL
LIN {X 0,Y 329.922,Z 322.861,A -85,B 0,C 180,E1 -15006.429,E2 -15006.429} C_VEL
LIN {X 0,Y 332.332,Z 326.359,A -85,B 0,C 180,E1 -15006.946,E2 -15006.946} C_VEL
LIN {X 0,Y 333.847,Z 328.148,A -85,B 0,C 180,E1 -15007.255,E2 -15007.255} C_VEL
LIN {X 0,Y 336.858,Z 331.835,A -85,B 0,C 180,E1 -15007.874,E2 -15007.874} C_VEL
LIN {X 0,Y 341.329,Z 337.18,A -85,B 0,C 180,E1 -15008.865,E2 -15008.865} C_VEL
LIN {X 0,Y 343.577,Z 339.682,A -85,B 0,C 180,E1 -15009.36,E2 -15009.36} C_VEL
LIN {X 0,Y 347.348,Z 343.653,A -85,B 0,C 180,E1 -15010.249,E2 -15010.249} C_VEL
LIN {X 0,Y 352.042,Z 348.766,A -85,B 0,C 180,E1 -15011.415,E2 -15011.415} C_VEL
LIN {X 0,Y 354.731,Z 351.21,A -85,B 0,C 180,E1 -15012.089,E2 -15012.089} C_VEL
LIN {X 0,Y 358.929,Z 355.424,A -85,B 0,C 180,E1 -15013.243,E2 -15013.243} C_VEL
LIN {X 0,Y 361.622,Z 357.669,A -85,B 0,C 180,E1 -15014.013,E2 -15014.013} C_VEL
LIN {X 0,Y 365.635,Z 361.687,A -85,B 0,C 180,E1 -15015.258,E2 -15015.258} C_VEL
LIN {X 0,Y 369.617,Z 364.847,A -85,B 0,C 180,E1 -15016.584,E2 -15016.584} C_VEL
LIN {X 0,Y 373.295,Z 368.422,A -85,B 0,C 180,E1 -15017.979,E2 -15017.979} C_VEL
LIN {X 0,Y 377.095,Z 371.047,A -85,B 0,C 180,E1 -15019.567,E2 -15019.567} C_VEL
LIN {X 0,Y 378.503,Z 371.984,A -85,B 0,C 180,E1 -15020.245,E2 -15020.245} C_VEL
LIN {X 0,Y 381.112,Z 374.829,A -85,B 0,C 180,E1 -15021.67,E2 -15021.67} C_VEL
LIN {X 0,Y 383.334,Z 376.638,A -85,B 0,C 180,E1 -15023.062,E2 -15023.062} C_VEL
LIN {X 0,Y 385.526,Z 377.999,A -85,B 0,C 180,E1 -15024.77,E2 -15024.77} C_VEL
LIN {X 0,Y 387.235,Z 378.642,A -85,B 0,C 180,E1 -15026.554,E2 -15026.554} C_VEL
LIN {X 0,Y 388.257,Z 379.202,A -85,B 0,C 180,E1 -15028.444,E2 -15028.444} C_VEL
LIN {X 0,Y 388.542,Z 379.227,A -85,B 0,C 180,E1 -15030,E2 -15030} C_VEL
LIN {X 0,Y 388.257,Z 379.184,A -85,B 0,C 180,E1 -15031.556,E2 -15031.556} C_VEL
LIN {X 0,Y 387.234,Z 378.67,A -85,B 0,C 180,E1 -15033.443,E2 -15033.443} C_VEL
LIN {X 0,Y 385.526,Z 378,A -85,B 0,C 180,E1 -15035.23,E2 -15035.23} C_VEL
LIN {X 0,Y 383.278,Z 376.595,A -85,B 0,C 180,E1 -15036.977,E2 -15036.977} C_VEL
LIN {X 0,Y 380.599,Z 374.308,A -85,B 0,C 180,E1 -15038.639,E2 -15038.639} C_VEL
LIN {X 0,Y 377.707,Z 371.348,A -85,B 0,C 180,E1 -15040.146,E2 -15040.146} C_VEL
LIN {X 0,Y 373.851,Z 368.917,A -85,B 0,C 180,E1 -15041.791,E2 -15041.791} C_VEL
LIN {X 0,Y 369.775,Z 365.065,A -85,B 0,C 180,E1 -15043.355,E2 -15043.355} C_VEL
LIN {X 0,Y 367.883,Z 363.434,A -85,B 0,C 180,E1 -15043.999,E2 -15043.999} C_VEL
LIN {X 0,Y 363.711,Z 359.953,A -85,B 0,C 180,E1 -15045.341,E2 -15045.341} C_VEL
LIN {X 0,Y 360.454,Z 356.588,A -85,B 0,C 180,E1 -15046.335,E2 -15046.335} C_VEL
LIN {X 0,Y 356.027,Z 352.677,A -85,B 0,C 180,E1 -15047.557,E2 -15047.557} C_VEL
LIN {X 0,Y 353.026,Z 349.612,A -85,B 0,C 180,E1 -15048.342,E2 -15048.342} C_VEL
LIN {X 0,Y 349.006,Z 345.521,A -85,B 0,C 180,E1 -15049.361,E2 -15049.361} C_VEL
LIN {X 0,Y 346.947,Z 343.303,A -85,B 0,C 180,E1 -15049.842,E2 -15049.842} C_VEL
LIN {X 0,Y 343.168,Z 339.146,A -85,B 0,C 180,E1 -15050.737,E2 -15050.737} C_VEL
LIN {X 0,Y 338.397,Z 333.83,A -85,B 0,C 180,E1 -15051.778,E2 -15051.778} C_VEL
LIN {X 0,Y 336.613,Z 331.601,A -85,B 0,C 180,E1 -15052.177,E2 -15052.177} C_VEL
LIN {X 0,Y 333.567,Z 327.726,A -85,B 0,C 180,E1 -15052.804,E2 -15052.804} C_VEL
LIN {X 0,Y 330.473,Z 323.86,A -85,B 0,C 180,E1 -15053.449,E2 -15053.449} C_VEL
LIN {X 0,Y 329.168,Z 321.932,A -85,B 0,C 180,E1 -15053.716,E2 -15053.716} C_VEL
LIN {X 0,Y 327.279,Z 319.491,A -85,B 0,C 180,E1 -15054.079,E2 -15054.079} C_VEL
LIN {X 0,Y 326.716,Z 317.711,A -85,B 0,C 180,E1 -15054.334,E2 -15054.334} C_VEL
LIN {X 0,Y 326.683,Z 317.294,A -85,B 0,C 180,E1 -15054.803,E2 -15054.803} C_VEL
LIN {X 0,Y 326.644,Z 317.282,A -85,B 0,C 180,E1 -15058.251,E2 -15058.251} C_VEL
LIN {X 0,Y 326.584,Z 317.302,A -85,B 0,C 180,E1 -15061.095,E2 -15061.095} C_VEL
LIN {X 0,Y 326.601,Z 317.272,A -85,B 0,C 180,E1 -15064.019,E2 -15064.019} C_VEL
LIN {X 0,Y 326.624,Z 317.297,A -85,B 0,C 180,E1 -15067.239,E2 -15067.239} C_VEL
LIN {X 0,Y 326.596,Z 317.275,A -85,B 0,C 180,E1 -15070.207,E2 -15070.207} C_VEL
LIN {X 0,Y 326.579,Z 317.269,A -85,B 0,C 180,E1 -15073.521,E2 -15073.521} C_VEL
LIN {X 0,Y 326.62,Z 317.301,A -85,B 0,C 180,E1 -15077.018,E2 -15077.018} C_VEL
LIN {X 0,Y 326.638,Z 317.291,A -85,B 0,C 180,E1 -15080.766,E2 -15080.766} C_VEL
LIN {X 0,Y 326.605,Z 317.289,A -85,B 0,C 180,E1 -15084.48,E2 -15084.48} C_VEL
LIN {X 0,Y 326.602,Z 317.298,A -85,B 0,C 180,E1 -15087.456,E2 -15087.456} C_VEL
LIN {X 0,Y 326.653,Z 317.292,A -85,B 0,C 180,E1 -15090.341,E2 -15090.341} C_VEL
LIN {X 0,Y 326.682,Z 317.281,A -85,B 0,C 180,E1 -15094.516,E2 -15094.516} C_VEL
LIN {X 0,Y 326.638,Z 317.289,A -85,B 0,C 180,E1 -15098.546,E2 -15098.546} C_VEL
LIN {X 0,Y 326.737,Z 317.257,A -85,B 0,C 180,E1 -15101.178,E2 -15101.178} C_VEL
LIN {X 0,Y 326.75,Z 317.284,A -85,B 0,C 180,E1 -15105.286,E2 -15105.286} C_VEL
LIN {X 0,Y 326.1,Z 317.363,A -85,B 0,C 180,E1 -15106.315,E2 -15106.315} C_VEL
LIN {X 0,Y 323.233,Z 317.708,A -85,B 0,C 180,E1 -15107.989,E2 -15107.989} C_VEL
LIN {X 0,Y 320.824,Z 317.991,A -85,B 0,C 180,E1 -15109.346,E2 -15109.346} C_VEL
LIN {X 0,Y 319.839,Z 318.108,A -85,B 0,C 180,E1 -15110.397,E2 -15110.397} C_VEL
LIN {X 0,Y 319.786,Z 318.117,A -85,B 0,C 180,E1 -15110.752,E2 -15110.752} C_VEL
LIN {X 0,Y 319.936,Z 318.129,A -85,B 0,C 180,E1 -15113.695,E2 -15113.695} C_VEL
LIN {X 0,Y 319.982,Z 318.111,A -85,B 0,C 180,E1 -15117.483,E2 -15117.483} C_VEL
LIN {X 0,Y 320.124,Z 318.07,A -85,B 0,C 180,E1 -15120.001,E2 -15120.001} C_VEL
LIN {X 0,Y 319.983,Z 318.115,A -85,B 0,C 180,E1 -15122.518,E2 -15122.518} C_VEL
LIN {X 0,Y 319.936,Z 318.127,A -85,B 0,C 180,E1 -15126.306,E2 -15126.306} C_VEL
LIN {X 0,Y 319.831,Z 318.11,A -85,B 0,C 180,E1 -15128.849,E2 -15128.849} C_VEL
LIN {X 0,Y 319.675,Z 318.157,A -85,B 0,C 180,E1 -15132.701,E2 -15132.701} C_VEL
LIN {X 0,Y 319.694,Z 318.155,A -85,B 0,C 180,E1 -15135.296,E2 -15135.296} C_VEL
LIN {X 0,Y 319.646,Z 318.139,A -85,B 0,C 180,E1 -15139.257,E2 -15139.257} C_VEL
LIN {X 0,Y 319.555,Z 318.176,A -85,B 0,C 180,E1 -15143.321,E2 -15143.321} C_VEL
LIN {X 0,Y 319.613,Z 318.149,A -85,B 0,C 180,E1 -15146.091,E2 -15146.091} C_VEL
LIN {X 0,Y 319.576,Z 318.17,A -85,B 0,C 180,E1 -15148.936,E2 -15148.936} C_VEL
LIN {X 0,Y 319.526,Z 318.181,A -85,B 0,C 180,E1 -15151.863,E2 -15151.863} C_VEL
LIN {X 0,Y 319.575,Z 318.168,A -85,B 0,C 180,E1 -15155.544,E2 -15155.544} C_VEL
LIN {X 0,Y 319.556,Z 318.167,A -85,B 0,C 180,E1 -15159.67,E2 -15159.67} C_VEL
LIN {X 0,Y 319.519,Z 318.181,A -85,B 0,C 180,E1 -15163.462,E2 -15163.462} C_VEL
LIN {X 0,Y 319.55,Z 318.179,A -85,B 0,C 180,E1 -15167.017,E2 -15167.017} C_VEL
LIN {X 0,Y 319.513,Z 318.163,A -85,B 0,C 180,E1 -15170.367,E2 -15170.367} C_VEL
LIN {X 0,Y 319.555,Z 318.165,A -85,B 0,C 180,E1 -15173.573,E2 -15173.573} C_VEL
LIN {X 0,Y 319.62,Z 318.268,A -85,B 0,C 180,E1 -15176.001,E2 -15176.001} C_VEL
LIN {X 0,Y 320.995,Z 324.824,A -85,B 0,C 180,E1 -15178.638,E2 -15178.638} C_VEL
LIN {X 0,Y 322.752,Z 334.077,A -85,B 0,C 180,E1 -15182.085,E2 -15182.085} C_VEL
LIN {X 0,Y 323.129,Z 338.367,A -85,B 0,C 180,E1 -15183.654,E2 -15183.654} C_VEL
LIN {X 0,Y 322.658,Z 341.935,A -85,B 0,C 180,E1 -15184.832,E2 -15184.832} C_VEL
LIN {X 0,Y 323.545,Z 346.402,A -85,B 0,C 180,E1 -15185.08,E2 -15185.08} C_VEL
LIN {X 0,Y 328.553,Z 370.852,A -85,B 0,C 180,E1 -15186.055,E2 -15186.055} C_VEL
LIN {X 0,Y 330.65,Z 383.403,A -85,B 0,C 180,E1 -15186.506,E2 -15186.506} C_VEL
LIN {X 0,Y 329.257,Z 446.905,A -85,B 0,C 180,E1 -15187.902,E2 -15187.902} C_VEL
LIN {X 0,Y 328.651,Z 457.635,A -85,B 0,C 180,E1 -15188.272,E2 -15188.272} C_VEL
LIN {X 0,Y 327.997,Z 466.733,A -85,B 0,C 180,E1 -15188.721,E2 -15188.721} C_VEL
LIN {X 0,Y 326.985,Z 477.091,A -85,B 0,C 180,E1 -15189.394,E2 -15189.394} C_VEL
LIN {X 0,Y 325.988,Z 486.222,A -85,B 0,C 180,E1 -15190.151,E2 -15190.151} C_VEL
LIN {X 0,Y 324.89,Z 495.217,A -85,B 0,C 180,E1 -15191.066,E2 -15191.066} C_VEL
LIN {X 0,Y 323.705,Z 503.943,A -85,B 0,C 180,E1 -15192.142,E2 -15192.142} C_VEL
LIN {X 0,Y 322.703,Z 511.337,A -85,B 0,C 180,E1 -15193.228,E2 -15193.228} C_VEL
LIN {X 0,Y 321.692,Z 518.79,A -85,B 0,C 180,E1 -15194.524,E2 -15194.524} C_VEL
LIN {X 0,Y 320.876,Z 524.761,A -85,B 0,C 180,E1 -15195.736,E2 -15195.736} C_VEL
LIN {X 0,Y 319.833,Z 531.296,A -85,B 0,C 180,E1 -15197.307,E2 -15197.307} C_VEL
LIN {X 0,Y 319.206,Z 535.798,A -85,B 0,C 180,E1 -15198.571,E2 -15198.571} C_VEL
LIN {X 0,Y 318.543,Z 541.291,A -85,B 0,C 180,E1 -15200.476,E2 -15200.476} C_VEL
LIN {X 0,Y 318.079,Z 545.617,A -85,B 0,C 180,E1 -15202.382,E2 -15202.382} C_VEL
LIN {X 0,Y 317.84,Z 548.888,A -85,B 0,C 180,E1 -15204.291,E2 -15204.291} C_VEL
LIN {X 0,Y 317.786,Z 551.175,A -85,B 0,C 180,E1 -15206.196,E2 -15206.196} C_VEL
LIN {X 0,Y 317.756,Z 552.234,A -85,B 0,C 180,E1 -15207.465,E2 -15207.465} C_VEL
LIN {X 0,Y 317.734,Z 552.823,A -85,B 0,C 180,E1 -15208.733,E2 -15208.733} C_VEL
LIN {X 0,Y 317.734,Z 552.823,A -85,B 0,C 180,E1 -15211.267,E2 -15211.267} C_VEL
LIN {X 0,Y 317.756,Z 552.234,A -85,B 0,C 180,E1 -15212.535,E2 -15212.535} C_VEL
LIN {X 0,Y 317.796,Z 549.785,A -85,B 0,C 180,E1 -15215.075,E2 -15215.075} C_VEL
LIN {X 0,Y 317.985,Z 546.835,A -85,B 0,C 180,E1 -15216.982,E2 -15216.982} C_VEL
LIN {X 0,Y 318.366,Z 542.846,A -85,B 0,C 180,E1 -15218.889,E2 -15218.889} C_VEL
LIN {X 0,Y 318.957,Z 537.714,A -85,B 0,C 180,E1 -15220.794,E2 -15220.794} C_VEL
LIN {X 0,Y 319.64,Z 532.451,A -85,B 0,C 180,E1 -15222.379,E2 -15222.379} C_VEL
LIN {X 0,Y 320.649,Z 526.137,A -85,B 0,C 180,E1 -15223.951,E2 -15223.951} C_VEL
LIN {X 0,Y 321.462,Z 520.184,A -85,B 0,C 180,E1 -15225.209,E2 -15225.209} C_VEL
LIN {X 0,Y 322.409,Z 513.256,A -85,B 0,C 180,E1 -15226.462,E2 -15226.462} C_VEL
LIN {X 0,Y 323.547,Z 505.077,A -85,B 0,C 180,E1 -15227.704,E2 -15227.704} C_VEL
LIN {X 0,Y 324.738,Z 496.569,A -85,B 0,C 180,E1 -15228.779,E2 -15228.779} C_VEL
LIN {X 0,Y 325.865,Z 487.856,A -85,B 0,C 180,E1 -15229.693,E2 -15229.693} C_VEL
LIN {X 0,Y 326.898,Z 478.098,A -85,B 0,C 180,E1 -15230.53,E2 -15230.53} C_VEL
LIN {X 0,Y 327.882,Z 468.02,A -85,B 0,C 180,E1 -15231.205,E2 -15231.205} C_VEL
LIN {X 0,Y 328.562,Z 458.508,A -85,B 0,C 180,E1 -15231.693,E2 -15231.693} C_VEL
LIN {X 0,Y 329.206,Z 448.203,A -85,B 0,C 180,E1 -15232.061,E2 -15232.061} C_VEL
LIN {X 0,Y 330.231,Z 404.685,A -85,B 0,C 180,E1 -15233.033,E2 -15233.033} C_VEL
LIN {X 0,Y 330.487,Z 381.717,A -85,B 0,C 180,E1 -15233.545,E2 -15233.545} C_VEL
LIN {X 0,Y 325.49,Z 355.221,A -85,B 0,C 180,E1 -15234.553,E2 -15234.553} C_VEL
LIN {X 0,Y 322.676,Z 342.263,A -85,B 0,C 180,E1 -15235.122,E2 -15235.122} C_VEL
LIN {X 0,Y 322.802,Z 340.769,A -85,B 0,C 180,E1 -15235.501,E2 -15235.501} C_VEL
LIN {X 0,Y 323.133,Z 336.814,A -85,B 0,C 180,E1 -15236.907,E2 -15236.907} C_VEL
LIN {X 0,Y 321.937,Z 329.601,A -85,B 0,C 180,E1 -15239.603,E2 -15239.603} C_VEL
LIN {X 0,Y 319.966,Z 319.975,A -85,B 0,C 180,E1 -15243.306,E2 -15243.306} C_VEL
LIN {X 0,Y 319.59,Z 318.187,A -85,B 0,C 180,E1 -15244.107,E2 -15244.107} C_VEL
LIN {X 0,Y 319.532,Z 318.185,A -85,B 0,C 180,E1 -15248.013,E2 -15248.013} C_VEL
LIN {X 0,Y 319.503,Z 318.165,A -85,B 0,C 180,E1 -15251.592,E2 -15251.592} C_VEL
LIN {X 0,Y 319.486,Z 318.185,A -85,B 0,C 180,E1 -15254.742,E2 -15254.742} C_VEL
LIN {X 0,Y 319.523,Z 318.181,A -85,B 0,C 180,E1 -15258.402,E2 -15258.402} C_VEL
LIN {X 0,Y 319.54,Z 318.181,A -85,B 0,C 180,E1 -15261.987,E2 -15261.987} C_VEL
LIN {X 0,Y 319.555,Z 318.164,A -85,B 0,C 180,E1 -15265.122,E2 -15265.122} C_VEL
LIN {X 0,Y 319.562,Z 318.178,A -85,B 0,C 180,E1 -15269.058,E2 -15269.058} C_VEL
LIN {X 0,Y 319.601,Z 318.151,A -85,B 0,C 180,E1 -15272.497,E2 -15272.497} C_VEL
LIN {X 0,Y 319.597,Z 318.163,A -85,B 0,C 180,E1 -15275.303,E2 -15275.303} C_VEL
LIN {X 0,Y 319.596,Z 318.158,A -85,B 0,C 180,E1 -15279.399,E2 -15279.399} C_VEL
LIN {X 0,Y 319.652,Z 318.138,A -85,B 0,C 180,E1 -15282.072,E2 -15282.072} C_VEL
LIN {X 0,Y 319.726,Z 318.155,A -85,B 0,C 180,E1 -15286.007,E2 -15286.007} C_VEL
LIN {X 0,Y 319.746,Z 318.12,A -85,B 0,C 180,E1 -15289.872,E2 -15289.872} C_VEL
LIN {X 0,Y 319.906,Z 318.12,A -85,B 0,C 180,E1 -15292.425,E2 -15292.425} C_VEL
LIN {X 0,Y 319.739,Z 318.156,A -85,B 0,C 180,E1 -15294.955,E2 -15294.955} C_VEL
LIN {X 0,Y 319.983,Z 318.115,A -85,B 0,C 180,E1 -15297.482,E2 -15297.482} C_VEL
LIN {X 0,Y 320.124,Z 318.07,A -85,B 0,C 180,E1 -15299.999,E2 -15299.999} C_VEL
LIN {X 0,Y 319.982,Z 318.111,A -85,B 0,C 180,E1 -15302.517,E2 -15302.517} C_VEL
LIN {X 0,Y 319.911,Z 318.127,A -85,B 0,C 180,E1 -15306.655,E2 -15306.655} C_VEL
LIN {X 0,Y 319.744,Z 318.119,A -85,B 0,C 180,E1 -15310.127,E2 -15310.127} C_VEL
LIN {X 0,Y 319.723,Z 318.159,A -85,B 0,C 180,E1 -15314.724,E2 -15314.724} C_VEL
LIN {X 0,Y 319.681,Z 318.134,A -85,B 0,C 180,E1 -15319.037,E2 -15319.037} C_VEL
LIN {X 0,Y 319.562,Z 318.179,A -85,B 0,C 180,E1 -15323.319,E2 -15323.319} C_VEL
LIN {X 0,Y 319.627,Z 318.155,A -85,B 0,C 180,E1 -15326.088,E2 -15326.088} C_VEL
LIN {X 0,Y 319.582,Z 318.162,A -85,B 0,C 180,E1 -15328.933,E2 -15328.933} C_VEL
LIN {X 0,Y 319.526,Z 318.182,A -85,B 0,C 180,E1 -15331.861,E2 -15331.861} C_VEL
LIN {X 0,Y 319.572,Z 318.165,A -85,B 0,C 180,E1 -15335.543,E2 -15335.543} C_VEL
LIN {X 0,Y 319.592,Z 318.176,A -85,B 0,C 180,E1 -15338.004,E2 -15338.004} C_VEL
LIN {X 0,Y 319.589,Z 318.166,A -85,B 0,C 180,E1 -15341.611,E2 -15341.611} C_VEL
LIN {X 0,Y 319.558,Z 318.167,A -85,B 0,C 180,E1 -15345.271,E2 -15345.271} C_VEL
LIN {X 0,Y 319.527,Z 318.137,A -85,B 0,C 180,E1 -15348.713,E2 -15348.713} C_VEL
LIN {X 0,Y 319.591,Z 318.178,A -85,B 0,C 180,E1 -15352.34,E2 -15352.34} C_VEL
LIN {X 0,Y 319.554,Z 318.147,A -85,B 0,C 180,E1 -15355.124,E2 -15355.124} C_VEL
LIN {X 0,Y 319.561,Z 318.173,A -85,B 0,C 180,E1 -15359.059,E2 -15359.059} C_VEL
LIN {X 0,Y 319.6,Z 318.172,A -85,B 0,C 180,E1 -15362.498,E2 -15362.498} C_VEL
LIN {X 0,Y 319.674,Z 318.393,A -85,B 0,C 180,E1 -15364.615,E2 -15364.615} C_VEL
LIN {X 0,Y 319.929,Z 319.398,A -85,B 0,C 180,E1 -15364.85,E2 -15364.85} C_VEL
LIN {X 0,Y 321.437,Z 322.037,A -85,B 0,C 180,E1 -15365.149,E2 -15365.149} C_VEL
LIN {X 0,Y 322.642,Z 323.824,A -85,B 0,C 180,E1 -15365.36,E2 -15365.36} C_VEL
LIN {X 0,Y 325.151,Z 327.269,A -85,B 0,C 180,E1 -15365.823,E2 -15365.823} C_VEL
LIN {X 0,Y 328.94,Z 332.148,A -85,B 0,C 180,E1 -15366.545,E2 -15366.545} C_VEL
LIN {X 0,Y 333.498,Z 337.645,A -85,B 0,C 180,E1 -15367.473,E2 -15367.473} C_VEL
LIN {X 0,Y 337.941,Z 342.865,A -85,B 0,C 180,E1 -15368.415,E2 -15368.415} C_VEL
LIN {X 0,Y 343.657,Z 348.992,A -85,B 0,C 180,E1 -15369.675,E2 -15369.675} C_VEL
LIN {X 0,Y 346.502,Z 352.019,A -85,B 0,C 180,E1 -15370.345,E2 -15370.345} C_VEL
LIN {X 0,Y 350.729,Z 356.071,A -85,B 0,C 180,E1 -15371.37,E2 -15371.37} C_VEL
LIN {X 0,Y 355.887,Z 361.186,A -85,B 0,C 180,E1 -15372.714,E2 -15372.714} C_VEL
LIN {X 0,Y 359.776,Z 364.48,A -85,B 0,C 180,E1 -15373.784,E2 -15373.784} C_VEL
LIN {X 0,Y 364.217,Z 368.695,A -85,B 0,C 180,E1 -15375.14,E2 -15375.14} C_VEL
LIN {X 0,Y 367.715,Z 371.436,A -85,B 0,C 180,E1 -15376.28,E2 -15376.28} C_VEL
LIN {X 0,Y 371.643,Z 375.122,A -85,B 0,C 180,E1 -15377.722,E2 -15377.722} C_VEL
LIN {X 0,Y 375.541,Z 377.821,A -85,B 0,C 180,E1 -15379.301,E2 -15379.301} C_VEL
LIN {X 0,Y 377.239,Z 378.933,A -85,B 0,C 180,E1 -15380.082,E2 -15380.082} C_VEL
LIN {X 0,Y 380.028,Z 381.858,A -85,B 0,C 180,E1 -15381.569,E2 -15381.569} C_VEL
LIN {X 0,Y 382.58,Z 383.843,A -85,B 0,C 180,E1 -15383.16,E2 -15383.16} C_VEL
LIN {X 0,Y 384.954,Z 385.19,A -85,B 0,C 180,E1 -15385.034,E2 -15385.034} C_VEL
LIN {X 0,Y 386.611,Z 385.76,A -85,B 0,C 180,E1 -15386.874,E2 -15386.874} C_VEL
LIN {X 0,Y 387.517,Z 386.337,A -85,B 0,C 180,E1 -15388.961,E2 -15388.961} C_VEL
LIN {X 0,Y 387.677,Z 386.274,A -85,B 0,C 180,E1 -15390,E2 -15390} C_VEL
LIN {X 0,Y 387.389,Z 386.232,A -85,B 0,C 180,E1 -15391.559,E2 -15391.559} C_VEL
LIN {X 0,Y 386.606,Z 385.79,A -85,B 0,C 180,E1 -15393.126,E2 -15393.126} C_VEL
LIN {X 0,Y 384.954,Z 385.194,A -85,B 0,C 180,E1 -15394.966,E2 -15394.966} C_VEL
LIN {X 0,Y 382.579,Z 383.847,A -85,B 0,C 180,E1 -15396.84,E2 -15396.84} C_VEL
LIN {X 0,Y 379.894,Z 381.74,A -85,B 0,C 180,E1 -15398.511,E2 -15398.511} C_VEL
LIN {X 0,Y 376.433,Z 378.258,A -85,B 0,C 180,E1 -15400.316,E2 -15400.316} C_VEL
LIN {X 0,Y 372.429,Z 375.742,A -85,B 0,C 180,E1 -15401.98,E2 -15401.98} C_VEL
LIN {X 0,Y 368.258,Z 371.965,A -85,B 0,C 180,E1 -15403.536,E2 -15403.536} C_VEL
LIN {X 0,Y 365.954,Z 369.988,A -85,B 0,C 180,E1 -15404.304,E2 -15404.304} C_VEL
LIN {X 0,Y 361.521,Z 366.325,A -85,B 0,C 180,E1 -15405.683,E2 -15405.683} C_VEL
LIN {X 0,Y 358.079,Z 362.926,A -85,B 0,C 180,E1 -15406.696,E2 -15406.696} C_VEL
LIN {X 0,Y 353.449,Z 358.852,A -85,B 0,C 180,E1 -15407.942,E2 -15407.942} C_VEL
LIN {X 0,Y 350.236,Z 355.682,A -85,B 0,C 180,E1 -15408.753,E2 -15408.753} C_VEL
LIN {X 0,Y 346.198,Z 351.685,A -85,B 0,C 180,E1 -15409.726,E2 -15409.726} C_VEL
LIN {X 0,Y 342.977,Z 348.297,A -85,B 0,C 180,E1 -15410.485,E2 -15410.485} C_VEL
LIN {X 0,Y 335.086,Z 339.635,A -85,B 0,C 180,E1 -15412.201,E2 -15412.201} C_VEL
LIN {X 0,Y 329.947,Z 333.281,A -85,B 0,C 180,E1 -15413.26,E2 -15413.26} C_VEL
LIN {X 0,Y 326.379,Z 328.938,A -85,B 0,C 180,E1 -15413.941,E2 -15413.941} C_VEL
LIN {X 0,Y 322.763,Z 324.03,A -85,B 0,C 180,E1 -15414.619,E2 -15414.619} C_VEL
LIN {X 0,Y 321.437,Z 322.048,A -85,B 0,C 180,E1 -15414.851,E2 -15414.851} C_VEL
LIN {X 0,Y 319.917,Z 319.438,A -85,B 0,C 180,E1 -15415.145,E2 -15415.145} C_VEL
LIN {X 0,Y 319.674,Z 318.38,A -85,B 0,C 180,E1 -15415.385,E2 -15415.385} C_VEL
LIN {X 0,Y 319.574,Z 318.156,A -85,B 0,C 180,E1 -15418.934,E2 -15418.934} C_VEL
LIN {X 0,Y 319.525,Z 318.185,A -85,B 0,C 180,E1 -15421.862,E2 -15421.862} C_VEL
LIN {X 0,Y 319.574,Z 318.149,A -85,B 0,C 180,E1 -15425.543,E2 -15425.543} C_VEL
LIN {X 0,Y 319.575,Z 318.179,A -85,B 0,C 180,E1 -15428.007,E2 -15428.007} C_VEL
LIN {X 0,Y 319.524,Z 318.135,A -85,B 0,C 180,E1 -15431.598,E2 -15431.598} C_VEL
LIN {X 0,Y 319.564,Z 318.17,A -85,B 0,C 180,E1 -15435.272,E2 -15435.272} C_VEL
LIN {X 0,Y 319.572,Z 318.165,A -85,B 0,C 180,E1 -15438.72,E2 -15438.72} C_VEL
LIN {X 0,Y 319.591,Z 318.176,A -85,B 0,C 180,E1 -15442.339,E2 -15442.339} C_VEL
LIN {X 0,Y 319.552,Z 318.162,A -85,B 0,C 180,E1 -15445.123,E2 -15445.123} C_VEL
LIN {X 0,Y 319.563,Z 318.182,A -85,B 0,C 180,E1 -15449.058,E2 -15449.058} C_VEL
LIN {X 0,Y 319.601,Z 318.149,A -85,B 0,C 180,E1 -15452.498,E2 -15452.498} C_VEL
LIN {X 0,Y 319.597,Z 318.171,A -85,B 0,C 180,E1 -15455.304,E2 -15455.304} C_VEL
LIN {X 0,Y 319.589,Z 318.17,A -85,B 0,C 180,E1 -15458.048,E2 -15458.048} C_VEL
LIN {X 0,Y 319.681,Z 318.134,A -85,B 0,C 180,E1 -15460.963,E2 -15460.963} C_VEL
LIN {X 0,Y 319.723,Z 318.159,A -85,B 0,C 180,E1 -15465.278,E2 -15465.278} C_VEL
LIN {X 0,Y 319.744,Z 318.119,A -85,B 0,C 180,E1 -15469.873,E2 -15469.873} C_VEL
LIN {X 0,Y 319.786,Z 318.117,A -85,B 0,C 180,E1 -15470.752,E2 -15470.752} C_VEL
LIN {X 0,Y 319.509,Z 318.161,A -85,B 0,C 180,E1 -15471.456,E2 -15471.456} C_VEL
LIN {X 0,Y 317.539,Z 318.423,A -85,B 0,C 180,E1 -15472.834,E2 -15472.834} C_VEL
LIN {X 0,Y 313.739,Z 318.909,A -85,B 0,C 180,E1 -15474.899,E2 -15474.899} C_VEL
LIN {X 0,Y 312.75,Z 319.026,A -85,B 0,C 180,E1 -15475.974,E2 -15475.974} C_VEL
LIN {X 0,Y 312.713,Z 319.026,A -85,B 0,C 180,E1 -15476.338,E2 -15476.338} C_VEL
LIN {X 0,Y 312.982,Z 318.964,A -85,B 0,C 180,E1 -15478.714,E2 -15478.714} C_VEL
LIN {X 0,Y 312.983,Z 318.973,A -85,B 0,C 180,E1 -15481.287,E2 -15481.287} C_VEL
LIN {X 0,Y 312.709,Z 319.031,A -85,B 0,C 180,E1 -15485.158,E2 -15485.158} C_VEL
LIN {X 0,Y 312.846,Z 318.994,A -85,B 0,C 180,E1 -15487.747,E2 -15487.747} C_VEL
LIN {X 0,Y 312.663,Z 319.024,A -85,B 0,C 180,E1 -15491.672,E2 -15491.672} C_VEL
LIN {X 0,Y 312.694,Z 319.029,A -85,B 0,C 180,E1 -15494.888,E2 -15494.888} C_VEL
LIN {X 0,Y 312.604,Z 319.015,A -85,B 0,C 180,E1 -15499.226,E2 -15499.226} C_VEL
LIN {X 0,Y 312.521,Z 319.055,A -85,B 0,C 180,E1 -15502.781,E2 -15502.781} C_VEL
LIN {X 0,Y 312.592,Z 319.024,A -85,B 0,C 180,E1 -15505.934,E2 -15505.934} C_VEL
LIN {X 0,Y 312.534,Z 319.051,A -85,B 0,C 180,E1 -15509.652,E2 -15509.652} C_VEL
LIN {X 0,Y 312.516,Z 319.037,A -85,B 0,C 180,E1 -15513.69,E2 -15513.69} C_VEL
LIN {X 0,Y 312.516,Z 319.056,A -85,B 0,C 180,E1 -15517.387,E2 -15517.387} C_VEL
LIN {X 0,Y 312.488,Z 319.051,A -85,B 0,C 180,E1 -15520.71,E2 -15520.71} C_VEL
LIN {X 0,Y 312.449,Z 319.057,A -85,B 0,C 180,E1 -15524.211,E2 -15524.211} C_VEL
LIN {X 0,Y 312.454,Z 319.049,A -85,B 0,C 180,E1 -15527.926,E2 -15527.926} C_VEL
LIN {X 0,Y 312.484,Z 319.062,A -85,B 0,C 180,E1 -15531.923,E2 -15531.923} C_VEL
LIN {X 0,Y 312.551,Z 319.173,A -85,B 0,C 180,E1 -15535.553,E2 -15535.553} C_VEL
LIN {X 0,Y 313.978,Z 325.804,A -85,B 0,C 180,E1 -15538.276,E2 -15538.276} C_VEL
LIN {X 0,Y 315.524,Z 333.866,A -85,B 0,C 180,E1 -15541.388,E2 -15541.388} C_VEL
LIN {X 0,Y 316.166,Z 338.616,A -85,B 0,C 180,E1 -15543.194,E2 -15543.194} C_VEL
LIN {X 0,Y 315.915,Z 341.755,A -85,B 0,C 180,E1 -15544.26,E2 -15544.26} C_VEL
LIN {X 0,Y 316.919,Z 346.703,A -85,B 0,C 180,E1 -15544.535,E2 -15544.535} C_VEL
LIN {X 0,Y 322.247,Z 372.931,A -85,B 0,C 180,E1 -15545.61,E2 -15545.61} C_VEL
LIN {X 0,Y 324.047,Z 383.765,A -85,B 0,C 180,E1 -15546.011,E2 -15546.011} C_VEL
LIN {X 0,Y 322.699,Z 446.718,A -85,B 0,C 180,E1 -15547.428,E2 -15547.428} C_VEL
LIN {X 0,Y 322.057,Z 457.44,A -85,B 0,C 180,E1 -15547.803,E2 -15547.803} C_VEL
LIN {X 0,Y 321.386,Z 466.539,A -85,B 0,C 180,E1 -15548.261,E2 -15548.261} C_VEL
LIN {X 0,Y 320.34,Z 476.897,A -85,B 0,C 180,E1 -15548.946,E2 -15548.946} C_VEL
LIN {X 0,Y 319.318,Z 486.028,A -85,B 0,C 180,E1 -15549.718,E2 -15549.718} C_VEL
LIN {X 0,Y 318.181,Z 495.023,A -85,B 0,C 180,E1 -15550.652,E2 -15550.652} C_VEL
LIN {X 0,Y 316.955,Z 503.749,A -85,B 0,C 180,E1 -15551.748,E2 -15551.748} C_VEL
LIN {X 0,Y 315.898,Z 511.143,A -85,B 0,C 180,E1 -15552.856,E2 -15552.856} C_VEL
LIN {X 0,Y 314.818,Z 518.76,A -85,B 0,C 180,E1 -15554.211,E2 -15554.211} C_VEL
LIN {X 0,Y 313.743,Z 525.942,A -85,B 0,C 180,E1 -15555.735,E2 -15555.735} C_VEL
LIN {X 0,Y 312.68,Z 532.256,A -85,B 0,C 180,E1 -15557.341,E2 -15557.341} C_VEL
LIN {X 0,Y 311.957,Z 537.52,A -85,B 0,C 180,E1 -15558.96,E2 -15558.96} C_VEL
LIN {X 0,Y 311.341,Z 542.651,A -85,B 0,C 180,E1 -15560.909,E2 -15560.909} C_VEL
LIN {X 0,Y 310.922,Z 546.64,A -85,B 0,C 180,E1 -15562.859,E2 -15562.859} C_VEL
LIN {X 0,Y 310.706,Z 549.591,A -85,B 0,C 180,E1 -15564.809,E2 -15564.809} C_VEL
LIN {X 0,Y 310.679,Z 552.04,A -85,B 0,C 180,E1 -15567.407,E2 -15567.407} C_VEL
LIN {X 0,Y 310.649,Z 552.629,A -85,B 0,C 180,E1 -15568.704,E2 -15568.704} C_VEL
LIN {X 0,Y 310.649,Z 552.629,A -85,B 0,C 180,E1 -15571.296,E2 -15571.296} C_VEL
LIN {X 0,Y 310.679,Z 552.04,A -85,B 0,C 180,E1 -15572.593,E2 -15572.593} C_VEL
LIN {X 0,Y 310.7,Z 549.591,A -85,B 0,C 180,E1 -15575.191,E2 -15575.191} C_VEL
LIN {X 0,Y 310.919,Z 546.64,A -85,B 0,C 180,E1 -15577.141,E2 -15577.141} C_VEL
LIN {X 0,Y 311.341,Z 542.651,A -85,B 0,C 180,E1 -15579.091,E2 -15579.091} C_VEL
LIN {X 0,Y 311.957,Z 537.52,A -85,B 0,C 180,E1 -15581.04,E2 -15581.04} C_VEL
LIN {X 0,Y 312.679,Z 532.256,A -85,B 0,C 180,E1 -15582.659,E2 -15582.659} C_VEL
LIN {X 0,Y 313.731,Z 525.942,A -85,B 0,C 180,E1 -15584.265,E2 -15584.265} C_VEL
LIN {X 0,Y 314.803,Z 518.794,A -85,B 0,C 180,E1 -15585.783,E2 -15585.783} C_VEL
LIN {X 0,Y 315.885,Z 511.143,A -85,B 0,C 180,E1 -15587.145,E2 -15587.145} C_VEL
LIN {X 0,Y 317.112,Z 502.614,A -85,B 0,C 180,E1 -15588.41,E2 -15588.41} C_VEL
LIN {X 0,Y 318.569,Z 492.32,A -85,B 0,C 180,E1 -15589.659,E2 -15589.659} C_VEL
LIN {X 0,Y 320.066,Z 479.919,A -85,B 0,C 180,E1 -15590.82,E2 -15590.82} C_VEL
LIN {X 0,Y 321.167,Z 469.114,A -85,B 0,C 180,E1 -15591.586,E2 -15591.586} C_VEL
LIN {X 0,Y 321.932,Z 459.188,A -85,B 0,C 180,E1 -15592.121,E2 -15592.121} C_VEL
LIN {X 0,Y 322.6,Z 449.341,A -85,B 0,C 180,E1 -15592.495,E2 -15592.495} C_VEL
LIN {X 0,Y 323.167,Z 428.314,A -85,B 0,C 180,E1 -15593.002,E2 -15593.002} C_VEL
LIN {X 0,Y 323.984,Z 382.697,A -85,B 0,C 180,E1 -15594.02,E2 -15594.02} C_VEL
LIN {X 0,Y 319.036,Z 356.465,A -85,B 0,C 180,E1 -15595.048,E2 -15595.048} C_VEL
LIN {X 0,Y 315.922,Z 342.088,A -85,B 0,C 180,E1 -15595.696,E2 -15595.696} C_VEL
LIN {X 0,Y 315.987,Z 340.665,A -85,B 0,C 180,E1 -15596.057,E2 -15596.057} C_VEL
LIN {X 0,Y 316.135,Z 337.501,A -85,B 0,C 180,E1 -15597.221,E2 -15597.221} C_VEL
LIN {X 0,Y 314.549,Z 328.904,A -85,B 0,C 180,E1 -15600.55,E2 -15600.55} C_VEL
LIN {X 0,Y 312.689,Z 319.76,A -85,B 0,C 180,E1 -15604.186,E2 -15604.186} C_VEL
LIN {X 0,Y 312.526,Z 319.057,A -85,B 0,C 180,E1 -15604.597,E2 -15604.597} C_VEL
LIN {X 0,Y 312.484,Z 319.062,A -85,B 0,C 180,E1 -15608.077,E2 -15608.077} C_VEL
LIN {X 0,Y 312.454,Z 319.049,A -85,B 0,C 180,E1 -15612.074,E2 -15612.074} C_VEL
LIN {X 0,Y 312.456,Z 319.057,A -85,B 0,C 180,E1 -15616.034,E2 -15616.034} C_VEL
LIN {X 0,Y 312.502,Z 319.045,A -85,B 0,C 180,E1 -15619.874,E2 -15619.874} C_VEL
LIN {X 0,Y 312.531,Z 319.048,A -85,B 0,C 180,E1 -15624.05,E2 -15624.05} C_VEL
LIN {X 0,Y 312.5,Z 319.046,A -85,B 0,C 180,E1 -15627.333,E2 -15627.333} C_VEL
LIN {X 0,Y 312.54,Z 319.042,A -85,B 0,C 180,E1 -15631.278,E2 -15631.278} C_VEL
LIN {X 0,Y 312.579,Z 319.034,A -85,B 0,C 180,E1 -15634.71,E2 -15634.71} C_VEL
LIN {X 0,Y 312.532,Z 319.046,A -85,B 0,C 180,E1 -15638.912,E2 -15638.912} C_VEL
LIN {X 0,Y 312.632,Z 319.009,A -85,B 0,C 180,E1 -15641.655,E2 -15641.655} C_VEL
LIN {X 0,Y 312.688,Z 319.034,A -85,B 0,C 180,E1 -15645.685,E2 -15645.685} C_VEL
LIN {X 0,Y 312.692,Z 319,A -85,B 0,C 180,E1 -15649.641,E2 -15649.641} C_VEL
LIN {X 0,Y 312.846,Z 318.994,A -85,B 0,C 180,E1 -15652.253,E2 -15652.253} C_VEL
LIN {X 0,Y 312.709,Z 319.031,A -85,B 0,C 180,E1 -15654.842,E2 -15654.842} C_VEL
LIN {X 0,Y 312.983,Z 318.973,A -85,B 0,C 180,E1 -15658.713,E2 -15658.713} C_VEL
LIN {X 0,Y 312.982,Z 318.964,A -85,B 0,C 180,E1 -15661.286,E2 -15661.286} C_VEL
LIN {X 0,Y 312.708,Z 319.035,A -85,B 0,C 180,E1 -15665.157,E2 -15665.157} C_VEL
LIN {X 0,Y 312.846,Z 319.001,A -85,B 0,C 180,E1 -15667.746,E2 -15667.746} C_VEL
LIN {X 0,Y 312.661,Z 319.016,A -85,B 0,C 180,E1 -15671.671,E2 -15671.671} C_VEL
LIN {X 0,Y 312.692,Z 319.037,A -85,B 0,C 180,E1 -15674.887,E2 -15674.887} C_VEL
LIN {X 0,Y 312.622,Z 319.013,A -85,B 0,C 180,E1 -15679.236,E2 -15679.236} C_VEL
LIN {X 0,Y 312.538,Z 319.053,A -85,B 0,C 180,E1 -15682.789,E2 -15682.789} C_VEL
LIN {X 0,Y 312.595,Z 319.033,A -85,B 0,C 180,E1 -15685.935,E2 -15685.935} C_VEL
LIN {X 0,Y 312.538,Z 319.05,A -85,B 0,C 180,E1 -15689.65,E2 -15689.65} C_VEL
LIN {X 0,Y 312.512,Z 319.042,A -85,B 0,C 180,E1 -15693.689,E2 -15693.689} C_VEL
LIN {X 0,Y 312.545,Z 319.054,A -85,B 0,C 180,E1 -15697.381,E2 -15697.381} C_VEL
LIN {X 0,Y 312.518,Z 319.041,A -85,B 0,C 180,E1 -15700.704,E2 -15700.704} C_VEL
LIN {X 0,Y 312.523,Z 319.054,A -85,B 0,C 180,E1 -15704.196,E2 -15704.196} C_VEL
LIN {X 0,Y 312.483,Z 319.009,A -85,B 0,C 180,E1 -15707.918,E2 -15707.918} C_VEL
LIN {X 0,Y 312.536,Z 319.055,A -85,B 0,C 180,E1 -15711.909,E2 -15711.909} C_VEL
LIN {X 0,Y 312.5,Z 319.026,A -85,B 0,C 180,E1 -15715.79,E2 -15715.79} C_VEL
LIN {X 0,Y 312.515,Z 319.054,A -85,B 0,C 180,E1 -15718.854,E2 -15718.854} C_VEL
LIN {X 0,Y 312.565,Z 319.036,A -85,B 0,C 180,E1 -15721.825,E2 -15721.825} C_VEL
LIN {X 0,Y 312.602,Z 319.219,A -85,B 0,C 180,E1 -15723.742,E2 -15723.742} C_VEL
LIN {X 0,Y 312.823,Z 320.119,A -85,B 0,C 180,E1 -15723.98,E2 -15723.98} C_VEL
LIN {X 0,Y 314.29,Z 322.855,A -85,B 0,C 180,E1 -15724.259,E2 -15724.259} C_VEL
LIN {X 0,Y 317.383,Z 327.465,A -85,B 0,C 180,E1 -15724.753,E2 -15724.753} C_VEL
LIN {X 0,Y 320.785,Z 332.275,A -85,B 0,C 180,E1 -15725.344,E2 -15725.344} C_VEL
LIN {X 0,Y 325.428,Z 337.937,A -85,B 0,C 180,E1 -15726.172,E2 -15726.172} C_VEL
LIN {X 0,Y 329.995,Z 343.32,A -85,B 0,C 180,E1 -15727.046,E2 -15727.046} C_VEL
LIN {X 0,Y 335.059,Z 349.051,A -85,B 0,C 180,E1 -15728.074,E2 -15728.074} C_VEL
LIN {X 0,Y 340.968,Z 355.258,A -85,B 0,C 180,E1 -15729.347,E2 -15729.347} C_VEL
LIN {X 0,Y 347.401,Z 361.734,A -85,B 0,C 180,E1 -15730.835,E2 -15730.835} C_VEL
LIN {X 0,Y 350.487,Z 364.681,A -85,B 0,C 180,E1 -15731.605,E2 -15731.605} C_VEL
LIN {X 0,Y 355.024,Z 368.752,A -85,B 0,C 180,E1 -15732.773,E2 -15732.773} C_VEL
LIN {X 0,Y 357.823,Z 371.22,A -85,B 0,C 180,E1 -15733.54,E2 -15733.54} C_VEL
LIN {X 0,Y 362.396,Z 375.382,A -85,B 0,C 180,E1 -15734.895,E2 -15734.895} C_VEL
LIN {X 0,Y 366.017,Z 378.21,A -85,B 0,C 180,E1 -15736.054,E2 -15736.054} C_VEL
LIN {X 0,Y 370.012,Z 381.855,A -85,B 0,C 180,E1 -15737.482,E2 -15737.482} C_VEL
LIN {X 0,Y 373.584,Z 384.339,A -85,B 0,C 180,E1 -15738.882,E2 -15738.882} C_VEL
LIN {X 0,Y 375.881,Z 385.805,A -85,B 0,C 180,E1 -15739.874,E2 -15739.874} C_VEL
LIN {X 0,Y 378.947,Z 388.88,A -85,B 0,C 180,E1 -15741.468,E2 -15741.468} C_VEL
LIN {X 0,Y 381.669,Z 390.909,A -85,B 0,C 180,E1 -15743.143,E2 -15743.143} C_VEL
LIN {X 0,Y 384.063,Z 392.24,A -85,B 0,C 180,E1 -15745.023,E2 -15745.023} C_VEL
LIN {X 0,Y 385.734,Z 392.807,A -85,B 0,C 180,E1 -15746.867,E2 -15746.867} C_VEL
LIN {X 0,Y 386.655,Z 393.383,A -85,B 0,C 180,E1 -15748.959,E2 -15748.959} C_VEL
LIN {X 0,Y 386.811,Z 393.321,A -85,B 0,C 180,E1 -15750,E2 -15750} C_VEL
LIN {X 0,Y 386.523,Z 393.255,A -85,B 0,C 180,E1 -15751.563,E2 -15751.563} C_VEL
LIN {X 0,Y 385.729,Z 392.835,A -85,B 0,C 180,E1 -15753.133,E2 -15753.133} C_VEL
LIN {X 0,Y 384.063,Z 392.243,A -85,B 0,C 180,E1 -15754.977,E2 -15754.977} C_VEL
LIN {X 0,Y 381.669,Z 390.911,A -85,B 0,C 180,E1 -15756.856,E2 -15756.856} C_VEL
LIN {X 0,Y 378.692,Z 388.654,A -85,B 0,C 180,E1 -15758.683,E2 -15758.683} C_VEL
LIN {X 0,Y 375.155,Z 385.183,A -85,B 0,C 180,E1 -15760.465,E2 -15760.465} C_VEL
LIN {X 0,Y 370.951,Z 382.586,A -85,B 0,C 180,E1 -15762.17,E2 -15762.17} C_VEL
LIN {X 0,Y 366.633,Z 378.798,A -85,B 0,C 180,E1 -15763.741,E2 -15763.741} C_VEL
LIN {X 0,Y 363.842,Z 376.447,A -85,B 0,C 180,E1 -15764.66,E2 -15764.66} C_VEL
LIN {X 0,Y 358.945,Z 372.374,A -85,B 0,C 180,E1 -15766.135,E2 -15766.135} C_VEL
LIN {X 0,Y 355.512,Z 369.145,A -85,B 0,C 180,E1 -15767.094,E2 -15767.094} C_VEL
LIN {X 0,Y 350.755,Z 364.981,A -85,B 0,C 180,E1 -15768.327,E2 -15768.327} C_VEL
LIN {X 0,Y 347.398,Z 361.746,A -85,B 0,C 180,E1 -15769.166,E2 -15769.166} C_VEL
LIN {X 0,Y 342.558,Z 356.838,A -85,B 0,C 180,E1 -15770.296,E2 -15770.296} C_VEL
LIN {X 0,Y 336.783,Z 350.914,A -85,B 0,C 180,E1 -15771.553,E2 -15771.553} C_VEL
LIN {X 0,Y 331.163,Z 344.752,A -85,B 0,C 180,E1 -15772.712,E2 -15772.712} C_VEL
LIN {X 0,Y 326.217,Z 338.86,A -85,B 0,C 180,E1 -15773.679,E2 -15773.679} C_VEL
LIN {X 0,Y 322.175,Z 333.957,A -85,B 0,C 180,E1 -15774.422,E2 -15774.422} C_VEL
LIN {X 0,Y 318.295,Z 328.888,A -85,B 0,C 180,E1 -15775.089,E2 -15775.089} C_VEL
LIN {X 0,Y 314.994,Z 323.92,A -85,B 0,C 180,E1 -15775.629,E2 -15775.629} C_VEL
LIN {X 0,Y 312.908,Z 320.404,A -85,B 0,C 180,E1 -15775.986,E2 -15775.986} C_VEL
LIN {X 0,Y 312.616,Z 319.336,A -85,B 0,C 180,E1 -15776.194,E2 -15776.194} C_VEL
LIN {X 0,Y 312.548,Z 319.055,A -85,B 0,C 180,E1 -15776.725,E2 -15776.725} C_VEL
LIN {X 0,Y 312.532,Z 319.033,A -85,B 0,C 180,E1 -15779.651,E2 -15779.651} C_VEL
LIN {X 0,Y 312.513,Z 319.029,A -85,B 0,C 180,E1 -15783.689,E2 -15783.689} C_VEL
LIN {X 0,Y 312.546,Z 319.052,A -85,B 0,C 180,E1 -15787.381,E2 -15787.381} C_VEL
LIN {X 0,Y 312.488,Z 319.019,A -85,B 0,C 180,E1 -15790.708,E2 -15790.708} C_VEL
LIN {X 0,Y 312.513,Z 319.031,A -85,B 0,C 180,E1 -15794.197,E2 -15794.197} C_VEL
LIN {X 0,Y 312.541,Z 319.047,A -85,B 0,C 180,E1 -15797.906,E2 -15797.906} C_VEL
LIN {X 0,Y 312.551,Z 319.053,A -85,B 0,C 180,E1 -15801.905,E2 -15801.905} C_VEL
LIN {X 0,Y 312.499,Z 319.04,A -85,B 0,C 180,E1 -15805.79,E2 -15805.79} C_VEL
LIN {X 0,Y 312.517,Z 319.058,A -85,B 0,C 180,E1 -15808.854,E2 -15808.854} C_VEL
LIN {X 0,Y 312.567,Z 319.028,A -85,B 0,C 180,E1 -15811.825,E2 -15811.825} C_VEL
LIN {X 0,Y 312.578,Z 319.039,A -85,B 0,C 180,E1 -15814.711,E2 -15814.711} C_VEL
LIN {X 0,Y 312.58,Z 319.045,A -85,B 0,C 180,E1 -15817.529,E2 -15817.529} C_VEL
LIN {X 0,Y 312.63,Z 319.016,A -85,B 0,C 180,E1 -15821.657,E2 -15821.657} C_VEL
LIN {X 0,Y 312.686,Z 319.034,A -85,B 0,C 180,E1 -15825.687,E2 -15825.687} C_VEL
LIN {X 0,Y 312.69,Z 318.997,A -85,B 0,C 180,E1 -15829.642,E2 -15829.642} C_VEL
LIN {X 0,Y 312.846,Z 319.001,A -85,B 0,C 180,E1 -15832.254,E2 -15832.254} C_VEL
LIN {X 0,Y 312.708,Z 319.035,A -85,B 0,C 180,E1 -15834.843,E2 -15834.843} C_VEL
LIN {X 0,Y 312.713,Z 319.026,A -85,B 0,C 180,E1 -15836.338,E2 -15836.338} C_VEL
LIN {X 0,Y 312.183,Z 319.083,A -85,B 0,C 180,E1 -15837.417,E2 -15837.417} C_VEL
LIN {X 0,Y 309.449,Z 319.406,A -85,B 0,C 180,E1 -15839.174,E2 -15839.174} C_VEL
LIN {X 0,Y 307.045,Z 319.706,A -85,B 0,C 180,E1 -15840.599,E2 -15840.599} C_VEL
LIN {X 0,Y 305.986,Z 319.852,A -85,B 0,C 180,E1 -15841.701,E2 -15841.701} C_VEL
LIN {X 0,Y 305.889,Z 319.863,A -85,B 0,C 180,E1 -15842.075,E2 -15842.075} C_VEL
LIN {X 0,Y 305.835,Z 319.878,A -85,B 0,C 180,E1 -15846.598,E2 -15846.598} C_VEL
LIN {X 0,Y 305.698,Z 319.866,A -85,B 0,C 180,E1 -15849.262,E2 -15849.262} C_VEL
LIN {X 0,Y 305.583,Z 319.916,A -85,B 0,C 180,E1 -15853.297,E2 -15853.297} C_VEL
LIN {X 0,Y 305.588,Z 319.909,A -85,B 0,C 180,E1 -15856.021,E2 -15856.021} C_VEL
LIN {X 0,Y 305.555,Z 319.894,A -85,B 0,C 180,E1 -15859.437,E2 -15859.437} C_VEL
LIN {X 0,Y 305.482,Z 319.93,A -85,B 0,C 180,E1 -15863.04,E2 -15863.04} C_VEL
LIN {X 0,Y 305.521,Z 319.902,A -85,B 0,C 180,E1 -15866.219,E2 -15866.219} C_VEL
LIN {X 0,Y 305.484,Z 319.926,A -85,B 0,C 180,E1 -15869.048,E2 -15869.048} C_VEL
LIN {X 0,Y 305.438,Z 319.933,A -85,B 0,C 180,E1 -15871.953,E2 -15871.953} C_VEL
LIN {X 0,Y 305.458,Z 319.921,A -85,B 0,C 180,E1 -15875.115,E2 -15875.115} C_VEL
LIN {X 0,Y 305.437,Z 319.932,A -85,B 0,C 180,E1 -15878.528,E2 -15878.528} C_VEL
LIN {X 0,Y 305.453,Z 319.936,A -85,B 0,C 180,E1 -15882.587,E2 -15882.587} C_VEL
LIN {X 0,Y 305.42,Z 319.943,A -85,B 0,C 180,E1 -15886.345,E2 -15886.345} C_VEL
LIN {X 0,Y 305.408,Z 319.914,A -85,B 0,C 180,E1 -15889.886,E2 -15889.886} C_VEL
LIN {X 0,Y 305.462,Z 319.919,A -85,B 0,C 180,E1 -15893.637,E2 -15893.637} C_VEL
LIN {X 0,Y 305.522,Z 320.138,A -85,B 0,C 180,E1 -15895.117,E2 -15895.117} C_VEL
LIN {X 0,Y 307.159,Z 327.678,A -85,B 0,C 180,E1 -15898.248,E2 -15898.248} C_VEL
LIN {X 0,Y 308.93,Z 337.179,A -85,B 0,C 180,E1 -15902.048,E2 -15902.048} C_VEL
LIN {X 0,Y 309.127,Z 341.291,A -85,B 0,C 180,E1 -15903.592,E2 -15903.592} C_VEL
LIN {X 0,Y 309.266,Z 342.59,A -85,B 0,C 180,E1 -15903.745,E2 -15903.745} C_VEL
LIN {X 0,Y 314.505,Z 367.016,A -85,B 0,C 180,E1 -15904.829,E2 -15904.829} C_VEL
LIN {X 0,Y 317.527,Z 384.506,A -85,B 0,C 180,E1 -15905.509,E2 -15905.509} C_VEL
LIN {X 0,Y 316.176,Z 446.532,A -85,B 0,C 180,E1 -15906.936,E2 -15906.936} C_VEL
LIN {X 0,Y 315.505,Z 457.247,A -85,B 0,C 180,E1 -15907.317,E2 -15907.317} C_VEL
LIN {X 0,Y 314.806,Z 466.345,A -85,B 0,C 180,E1 -15907.783,E2 -15907.783} C_VEL
LIN {X 0,Y 313.846,Z 475.696,A -85,B 0,C 180,E1 -15908.403,E2 -15908.403} C_VEL
LIN {X 0,Y 312.68,Z 485.835,A -85,B 0,C 180,E1 -15909.268,E2 -15909.268} C_VEL
LIN {X 0,Y 311.462,Z 494.828,A -85,B 0,C 180,E1 -15910.217,E2 -15910.217} C_VEL
LIN {X 0,Y 310.193,Z 503.554,A -85,B 0,C 180,E1 -15911.336,E2 -15911.336} C_VEL
LIN {X 0,Y 309.09,Z 510.948,A -85,B 0,C 180,E1 -15912.466,E2 -15912.466} C_VEL
LIN {X 0,Y 308.076,Z 518.029,A -85,B 0,C 180,E1 -15913.743,E2 -15913.743} C_VEL
LIN {X 0,Y 307.057,Z 524.371,A -85,B 0,C 180,E1 -15915.079,E2 -15915.079} C_VEL
LIN {X 0,Y 305.953,Z 530.907,A -85,B 0,C 180,E1 -15916.72,E2 -15916.72} C_VEL
LIN {X 0,Y 305.21,Z 535.408,A -85,B 0,C 180,E1 -15918.04,E2 -15918.04} C_VEL
LIN {X 0,Y 304.459,Z 540.901,A -85,B 0,C 180,E1 -15920.031,E2 -15920.031} C_VEL
LIN {X 0,Y 303.96,Z 545.228,A -85,B 0,C 180,E1 -15922.026,E2 -15922.026} C_VEL
LIN {X 0,Y 303.743,Z 547.596,A -85,B 0,C 180,E1 -15923.357,E2 -15923.357} C_VEL
LIN {X 0,Y 303.64,Z 549.397,A -85,B 0,C 180,E1 -15924.688,E2 -15924.688} C_VEL
LIN {X 0,Y 303.603,Z 551.847,A -85,B 0,C 180,E1 -15927.346,E2 -15927.346} C_VEL
LIN {X 0,Y 303.566,Z 552.435,A -85,B 0,C 180,E1 -15928.673,E2 -15928.673} C_VEL
LIN {X 0,Y 303.566,Z 552.435,A -85,B 0,C 180,E1 -15931.327,E2 -15931.327} C_VEL
LIN {X 0,Y 303.603,Z 551.847,A -85,B 0,C 180,E1 -15932.654,E2 -15932.654} C_VEL
LIN {X 0,Y 303.62,Z 549.396,A -85,B 0,C 180,E1 -15935.312,E2 -15935.312} C_VEL
LIN {X 0,Y 303.841,Z 546.445,A -85,B 0,C 180,E1 -15937.309,E2 -15937.309} C_VEL
LIN {X 0,Y 304.29,Z 542.456,A -85,B 0,C 180,E1 -15939.304,E2 -15939.304} C_VEL
LIN {X 0,Y 304.965,Z 537.325,A -85,B 0,C 180,E1 -15941.296,E2 -15941.296} C_VEL
LIN {X 0,Y 305.739,Z 532.062,A -85,B 0,C 180,E1 -15942.951,E2 -15942.951} C_VEL
LIN {X 0,Y 306.821,Z 525.747,A -85,B 0,C 180,E1 -15944.593,E2 -15944.593} C_VEL
LIN {X 0,Y 307.755,Z 519.796,A -85,B 0,C 180,E1 -15945.904,E2 -15945.904} C_VEL
LIN {X 0,Y 308.756,Z 512.867,A -85,B 0,C 180,E1 -15947.212,E2 -15947.212} C_VEL
LIN {X 0,Y 310.027,Z 504.689,A -85,B 0,C 180,E1 -15948.503,E2 -15948.503} C_VEL
LIN {X 0,Y 311.288,Z 496.18,A -85,B 0,C 180,E1 -15949.623,E2 -15949.623} C_VEL
LIN {X 0,Y 312.513,Z 487.467,A -85,B 0,C 180,E1 -15950.572,E2 -15950.572} C_VEL
LIN {X 0,Y 313.631,Z 477.71,A -85,B 0,C 180,E1 -15951.44,E2 -15951.44} C_VEL
LIN {X 0,Y 314.684,Z 467.632,A -85,B 0,C 180,E1 -15952.14,E2 -15952.14} C_VEL
LIN {X 0,Y 315.45,Z 458.121,A -85,B 0,C 180,E1 -15952.644,E2 -15952.644} C_VEL
LIN {X 0,Y 316.115,Z 447.816,A -85,B 0,C 180,E1 -15953.026,E2 -15953.026} C_VEL
LIN {X 0,Y 317.299,Z 398.184,A -85,B 0,C 180,E1 -15954.177,E2 -15954.177} C_VEL
LIN {X 0,Y 317.496,Z 383.79,A -85,B 0,C 180,E1 -15954.511,E2 -15954.511} C_VEL
LIN {X 0,Y 312.969,Z 359.389,A -85,B 0,C 180,E1 -15955.491,E2 -15955.491} C_VEL
LIN {X 0,Y 309.135,Z 341.911,A -85,B 0,C 180,E1 -15956.301,E2 -15956.301} C_VEL
LIN {X 0,Y 309.174,Z 340.465,A -85,B 0,C 180,E1 -15956.676,E2 -15956.676} C_VEL
LIN {X 0,Y 308.938,Z 337.176,A -85,B 0,C 180,E1 -15957.953,E2 -15957.953} C_VEL
LIN {X 0,Y 307.14,Z 327.685,A -85,B 0,C 180,E1 -15961.754,E2 -15961.754} C_VEL
LIN {X 0,Y 305.518,Z 319.981,A -85,B 0,C 180,E1 -15964.971,E2 -15964.971} C_VEL
LIN {X 0,Y 305.416,Z 319.936,A -85,B 0,C 180,E1 -15968.52,E2 -15968.52} C_VEL
LIN {X 0,Y 305.434,Z 319.932,A -85,B 0,C 180,E1 -15972.581,E2 -15972.581} C_VEL
LIN {X 0,Y 305.423,Z 319.935,A -85,B 0,C 180,E1 -15976.344,E2 -15976.344} C_VEL
LIN {X 0,Y 305.456,Z 319.923,A -85,B 0,C 180,E1 -15979.891,E2 -15979.891} C_VEL
LIN {X 0,Y 305.476,Z 319.931,A -85,B 0,C 180,E1 -15983.631,E2 -15983.631} C_VEL
LIN {X 0,Y 305.461,Z 319.916,A -85,B 0,C 180,E1 -15986.482,E2 -15986.482} C_VEL
LIN {X 0,Y 305.455,Z 319.938,A -85,B 0,C 180,E1 -15989.589,E2 -15989.589} C_VEL
LIN {X 0,Y 305.492,Z 319.906,A -85,B 0,C 180,E1 -15992.605,E2 -15992.605} C_VEL
LIN {X 0,Y 305.499,Z 319.921,A -85,B 0,C 180,E1 -15995.537,E2 -15995.537} C_VEL
LIN {X 0,Y 305.501,Z 319.909,A -85,B 0,C 180,E1 -15999.813,E2 -15999.813} C_VEL
LIN {X 0,Y 305.568,Z 319.896,A -85,B 0,C 180,E1 -16002.602,E2 -16002.602} C_VEL
LIN {X 0,Y 305.643,Z 319.91,A -85,B 0,C 180,E1 -16005.348,E2 -16005.348} C_VEL
LIN {X 0,Y 305.629,Z 319.881,A -85,B 0,C 180,E1 -16009.399,E2 -16009.399} C_VEL
LIN {X 0,Y 305.79,Z 319.869,A -85,B 0,C 180,E1 -16012.073,E2 -16012.073} C_VEL
LIN {X 0,Y 305.68,Z 319.906,A -85,B 0,C 180,E1 -16014.723,E2 -16014.723} C_VEL
LIN {X 0,Y 305.95,Z 319.848,A -85,B 0,C 180,E1 -16018.683,E2 -16018.683} C_VEL
LIN {X 0,Y 305.949,Z 319.84,A -85,B 0,C 180,E1 -16021.316,E2 -16021.316} C_VEL
LIN {X 0,Y 305.679,Z 319.909,A -85,B 0,C 180,E1 -16025.276,E2 -16025.276} C_VEL
LIN {X 0,Y 305.79,Z 319.879,A -85,B 0,C 180,E1 -16027.926,E2 -16027.926} C_VEL
LIN {X 0,Y 305.595,Z 319.9,A -85,B 0,C 180,E1 -16031.945,E2 -16031.945} C_VEL
LIN {X 0,Y 305.63,Z 319.916,A -85,B 0,C 180,E1 -16035.034,E2 -16035.034} C_VEL
LIN {X 0,Y 305.569,Z 319.891,A -85,B 0,C 180,E1 -16039.444,E2 -16039.444} C_VEL
LIN {X 0,Y 305.483,Z 319.934,A -85,B 0,C 180,E1 -16043.041,E2 -16043.041} C_VEL
LIN {X 0,Y 305.524,Z 319.908,A -85,B 0,C 180,E1 -16046.221,E2 -16046.221} C_VEL
LIN {X 0,Y 305.488,Z 319.918,A -85,B 0,C 180,E1 -16049.05,E2 -16049.05} C_VEL
LIN {X 0,Y 305.438,Z 319.938,A -85,B 0,C 180,E1 -16051.952,E2 -16051.952} C_VEL
LIN {X 0,Y 305.455,Z 319.918,A -85,B 0,C 180,E1 -16055.113,E2 -16055.113} C_VEL
LIN {X 0,Y 305.487,Z 319.932,A -85,B 0,C 180,E1 -16058.539,E2 -16058.539} C_VEL
LIN {X 0,Y 305.5,Z 319.928,A -85,B 0,C 180,E1 -16062.597,E2 -16062.597} C_VEL
LIN {X 0,Y 305.465,Z 319.897,A -85,B 0,C 180,E1 -16066.353,E2 -16066.353} C_VEL
LIN {X 0,Y 305.456,Z 319.905,A -85,B 0,C 180,E1 -16069.893,E2 -16069.893} C_VEL
LIN {X 0,Y 305.496,Z 319.914,A -85,B 0,C 180,E1 -16073.626,E2 -16073.626} C_VEL
LIN {X 0,Y 305.459,Z 319.909,A -85,B 0,C 180,E1 -16076.483,E2 -16076.483} C_VEL
LIN {X 0,Y 305.452,Z 319.921,A -85,B 0,C 180,E1 -16079.591,E2 -16079.591} C_VEL
LIN {X 0,Y 305.526,Z 320.086,A -85,B 0,C 180,E1 -16082.99,E2 -16082.99} C_VEL
LIN {X 0,Y 305.769,Z 321.076,A -85,B 0,C 180,E1 -16083.248,E2 -16083.248} C_VEL
LIN {X 0,Y 309.33,Z 327.353,A -85,B 0,C 180,E1 -16083.811,E2 -16083.811} C_VEL
LIN {X 0,Y 315.162,Z 335.84,A -85,B 0,C 180,E1 -16084.711,E2 -16084.711} C_VEL
LIN {X 0,Y 321.637,Z 343.505,A -85,B 0,C 180,E1 -16085.771,E2 -16085.771} C_VEL
LIN {X 0,Y 326.495,Z 349.086,A -85,B 0,C 180,E1 -16086.657,E2 -16086.657} C_VEL
LIN {X 0,Y 331.498,Z 354.669,A -85,B 0,C 180,E1 -16087.635,E2 -16087.635} C_VEL
LIN {X 0,Y 337.794,Z 361.177,A -85,B 0,C 180,E1 -16088.948,E2 -16088.948} C_VEL
LIN {X 0,Y 344.046,Z 367.403,A -85,B 0,C 180,E1 -16090.343,E2 -16090.343} C_VEL
LIN {X 0,Y 347.951,Z 370.991,A -85,B 0,C 180,E1 -16091.26,E2 -16091.26} C_VEL
LIN {X 0,Y 352.952,Z 375.339,A -85,B 0,C 180,E1 -16092.516,E2 -16092.516} C_VEL
LIN {X 0,Y 359.357,Z 381.114,A -85,B 0,C 180,E1 -16094.299,E2 -16094.299} C_VEL
LIN {X 0,Y 364.145,Z 384.811,A -85,B 0,C 180,E1 -16095.766,E2 -16095.766} C_VEL
LIN {X 0,Y 368.209,Z 388.442,A -85,B 0,C 180,E1 -16097.173,E2 -16097.173} C_VEL
LIN {X 0,Y 372.201,Z 391.202,A -85,B 0,C 180,E1 -16098.698,E2 -16098.698} C_VEL
LIN {X 0,Y 374.42,Z 392.551,A -85,B 0,C 180,E1 -16099.628,E2 -16099.628} C_VEL
LIN {X 0,Y 377.752,Z 395.772,A -85,B 0,C 180,E1 -16101.306,E2 -16101.306} C_VEL
LIN {X 0,Y 380.706,Z 397.938,A -85,B 0,C 180,E1 -16103.09,E2 -16103.09} C_VEL
LIN {X 0,Y 383.172,Z 399.286,A -85,B 0,C 180,E1 -16105.011,E2 -16105.011} C_VEL
LIN {X 0,Y 384.859,Z 399.828,A -85,B 0,C 180,E1 -16106.86,E2 -16106.86} C_VEL
LIN {X 0,Y 385.794,Z 400.43,A -85,B 0,C 180,E1 -16108.956,E2 -16108.956} C_VEL
LIN {X 0,Y 385.946,Z 400.367,A -85,B 0,C 180,E1 -16110,E2 -16110} C_VEL
LIN {X 0,Y 385.654,Z 400.303,A -85,B 0,C 180,E1 -16111.566,E2 -16111.566} C_VEL
LIN {X 0,Y 384.854,Z 399.864,A -85,B 0,C 180,E1 -16113.14,E2 -16113.14} C_VEL
LIN {X 0,Y 383.172,Z 399.289,A -85,B 0,C 180,E1 -16114.989,E2 -16114.989} C_VEL
LIN {X 0,Y 380.706,Z 397.936,A -85,B 0,C 180,E1 -16116.91,E2 -16116.91} C_VEL
LIN {X 0,Y 377.564,Z 395.649,A -85,B 0,C 180,E1 -16118.792,E2 -16118.792} C_VEL
LIN {X 0,Y 373.596,Z 391.973,A -85,B 0,C 180,E1 -16120.732,E2 -16120.732} C_VEL
LIN {X 0,Y 369.306,Z 389.309,A -85,B 0,C 180,E1 -16122.419,E2 -16122.419} C_VEL
LIN {X 0,Y 365.06,Z 385.723,A -85,B 0,C 180,E1 -16123.923,E2 -16123.923} C_VEL
LIN {X 0,Y 362.055,Z 383.13,A -85,B 0,C 180,E1 -16124.893,E2 -16124.893} C_VEL
LIN {X 0,Y 357.097,Z 379.173,A -85,B 0,C 180,E1 -16126.35,E2 -16126.35} C_VEL
LIN {X 0,Y 353.196,Z 375.53,A -85,B 0,C 180,E1 -16127.421,E2 -16127.421} C_VEL
LIN {X 0,Y 347.95,Z 371.007,A -85,B 0,C 180,E1 -16128.74,E2 -16128.74} C_VEL
LIN {X 0,Y 340.576,Z 363.99,A -85,B 0,C 180,E1 -16130.456,E2 -16130.456} C_VEL
LIN {X 0,Y 333.342,Z 356.559,A -85,B 0,C 180,E1 -16131.996,E2 -16131.996} C_VEL
LIN {X 0,Y 327.608,Z 350.408,A -85,B 0,C 180,E1 -16133.129,E2 -16133.129} C_VEL
LIN {X 0,Y 322.158,Z 344.084,A -85,B 0,C 180,E1 -16134.139,E2 -16134.139} C_VEL
LIN {X 0,Y 317.779,Z 338.928,A -85,B 0,C 180,E1 -16134.877,E2 -16134.877} C_VEL
LIN {X 0,Y 313.703,Z 333.801,A -85,B 0,C 180,E1 -16135.517,E2 -16135.517} C_VEL
LIN {X 0,Y 308.303,Z 325.823,A -85,B 0,C 180,E1 -16136.335,E2 -16136.335} C_VEL
LIN {X 0,Y 305.768,Z 321.079,A -85,B 0,C 180,E1 -16136.751,E2 -16136.751} C_VEL
LIN {X 0,Y 305.52,Z 320.055,A -85,B 0,C 180,E1 -16137.04,E2 -16137.04} C_VEL
LIN {X 0,Y 305.452,Z 319.921,A -85,B 0,C 180,E1 -16140.409,E2 -16140.409} C_VEL
LIN {X 0,Y 305.458,Z 319.903,A -85,B 0,C 180,E1 -16144.078,E2 -16144.078} C_VEL
LIN {X 0,Y 305.496,Z 319.922,A -85,B 0,C 180,E1 -16146.735,E2 -16146.735} C_VEL
LIN {X 0,Y 305.452,Z 319.896,A -85,B 0,C 180,E1 -16150.6,E2 -16150.6} C_VEL
LIN {X 0,Y 305.455,Z 319.915,A -85,B 0,C 180,E1 -16154.501,E2 -16154.501} C_VEL
LIN {X 0,Y 305.487,Z 319.924,A -85,B 0,C 180,E1 -16158.152,E2 -16158.152} C_VEL
LIN {X 0,Y 305.513,Z 319.931,A -85,B 0,C 180,E1 -16161.604,E2 -16161.604} C_VEL
LIN {X 0,Y 305.455,Z 319.918,A -85,B 0,C 180,E1 -16164.887,E2 -16164.887} C_VEL
LIN {X 0,Y 305.445,Z 319.937,A -85,B 0,C 180,E1 -16168.355,E2 -16168.355} C_VEL
LIN {X 0,Y 305.513,Z 319.913,A -85,B 0,C 180,E1 -16171.114,E2 -16171.114} C_VEL
LIN {X 0,Y 305.564,Z 319.908,A -85,B 0,C 180,E1 -16174.088,E2 -16174.088} C_VEL
LIN {X 0,Y 305.492,Z 319.923,A -85,B 0,C 180,E1 -16178.403,E2 -16178.403} C_VEL
LIN {X 0,Y 305.582,Z 319.89,A -85,B 0,C 180,E1 -16181.218,E2 -16181.218} C_VEL
LIN {X 0,Y 305.641,Z 319.913,A -85,B 0,C 180,E1 -16185.349,E2 -16185.349} C_VEL
LIN {X 0,Y 305.627,Z 319.878,A -85,B 0,C 180,E1 -16189.4,E2 -16189.4} C_VEL
LIN {X 0,Y 305.789,Z 319.879,A -85,B 0,C 180,E1 -16192.074,E2 -16192.074} C_VEL
LIN {X 0,Y 305.679,Z 319.909,A -85,B 0,C 180,E1 -16194.724,E2 -16194.724} C_VEL
LIN {X 0,Y 305.949,Z 319.84,A -85,B 0,C 180,E1 -16198.684,E2 -16198.684} C_VEL
LIN {X 0,Y 305.95,Z 319.848,A -85,B 0,C 180,E1 -16201.317,E2 -16201.317} C_VEL
LIN {X 0,Y 305.889,Z 319.863,A -85,B 0,C 180,E1 -16202.075,E2 -16202.075} C_VEL
LIN {X 0,Y 305.183,Z 319.967,A -85,B 0,C 180,E1 -16203.172,E2 -16203.172} C_VEL
LIN {X 0,Y 302.28,Z 320.331,A -85,B 0,C 180,E1 -16204.957,E2 -16204.957} C_VEL
LIN {X 0,Y 299.843,Z 320.627,A -85,B 0,C 180,E1 -16206.405,E2 -16206.405} C_VEL
LIN {X 0,Y 298.809,Z 320.745,A -85,B 0,C 180,E1 -16207.528,E2 -16207.528} C_VEL
LIN {X 0,Y 298.73,Z 320.745,A -85,B 0,C 180,E1 -16207.908,E2 -16207.908} C_VEL
LIN {X 0,Y 298.547,Z 320.784,A -85,B 0,C 180,E1 -16212.232,E2 -16212.232} C_VEL
LIN {X 0,Y 298.58,Z 320.786,A -85,B 0,C 180,E1 -16215.195,E2 -16215.195} C_VEL
LIN {X 0,Y 298.52,Z 320.768,A -85,B 0,C 180,E1 -16219.245,E2 -16219.245} C_VEL
LIN {X 0,Y 298.424,Z 320.808,A -85,B 0,C 180,E1 -16223.601,E2 -16223.601} C_VEL
LIN {X 0,Y 298.48,Z 320.777,A -85,B 0,C 180,E1 -16226.576,E2 -16226.576} C_VEL
LIN {X 0,Y 298.413,Z 320.81,A -85,B 0,C 180,E1 -16229.643,E2 -16229.643} C_VEL
LIN {X 0,Y 298.391,Z 320.801,A -85,B 0,C 180,E1 -16232.801,E2 -16232.801} C_VEL
LIN {X 0,Y 298.441,Z 320.81,A -85,B 0,C 180,E1 -16236.808,E2 -16236.808} C_VEL
LIN {X 0,Y 298.385,Z 320.811,A -85,B 0,C 180,E1 -16241.089,E2 -16241.089} C_VEL
LIN {X 0,Y 298.397,Z 320.813,A -85,B 0,C 180,E1 -16243.104,E2 -16243.104} C_VEL
LIN {X 0,Y 298.37,Z 320.818,A -85,B 0,C 180,E1 -16246.916,E2 -16246.916} C_VEL
LIN {X 0,Y 298.354,Z 320.805,A -85,B 0,C 180,E1 -16251.019,E2 -16251.019} C_VEL
LIN {X 0,Y 298.464,Z 320.91,A -85,B 0,C 180,E1 -16254.545,E2 -16254.545} C_VEL
LIN {X 0,Y 299.622,Z 326.429,A -85,B 0,C 180,E1 -16256.952,E2 -16256.952} C_VEL
LIN {X 0,Y 301.186,Z 334.291,A -85,B 0,C 180,E1 -16260.22,E2 -16260.22} C_VEL
LIN {X 0,Y 302.245,Z 340.784,A -85,B 0,C 180,E1 -16262.849,E2 -16262.849} C_VEL
LIN {X 0,Y 302.313,Z 341.668,A -85,B 0,C 180,E1 -16263.054,E2 -16263.054} C_VEL
LIN {X 0,Y 305.931,Z 357.47,A -85,B 0,C 180,E1 -16263.835,E2 -16263.835} C_VEL
LIN {X 0,Y 310.463,Z 381.448,A -85,B 0,C 180,E1 -16264.842,E2 -16264.842} C_VEL
LIN {X 0,Y 311.097,Z 387.26,A -85,B 0,C 180,E1 -16265.042,E2 -16265.042} C_VEL
LIN {X 0,Y 309.579,Z 447.622,A -85,B 0,C 180,E1 -16266.459,E2 -16266.459} C_VEL
LIN {X 0,Y 308.91,Z 457.927,A -85,B 0,C 180,E1 -16266.849,E2 -16266.849} C_VEL
LIN {X 0,Y 308.118,Z 467.439,A -85,B 0,C 180,E1 -16267.362,E2 -16267.362} C_VEL
LIN {X 0,Y 307.151,Z 476.51,A -85,B 0,C 180,E1 -16267.996,E2 -16267.996} C_VEL
LIN {X 0,Y 306.05,Z 485.641,A -85,B 0,C 180,E1 -16268.797,E2 -16268.797} C_VEL
LIN {X 0,Y 304.775,Z 494.634,A -85,B 0,C 180,E1 -16269.764,E2 -16269.764} C_VEL
LIN {X 0,Y 303.435,Z 503.359,A -85,B 0,C 180,E1 -16270.904,E2 -16270.904} C_VEL
LIN {X 0,Y 302.286,Z 510.753,A -85,B 0,C 180,E1 -16272.058,E2 -16272.058} C_VEL
LIN {X 0,Y 301.18,Z 518.174,A -85,B 0,C 180,E1 -16273.433,E2 -16273.433} C_VEL
LIN {X 0,Y 300.143,Z 524.176,A -85,B 0,C 180,E1 -16274.727,E2 -16274.727} C_VEL
LIN {X 0,Y 299.022,Z 530.712,A -85,B 0,C 180,E1 -16276.407,E2 -16276.407} C_VEL
LIN {X 0,Y 298.233,Z 535.213,A -85,B 0,C 180,E1 -16277.755,E2 -16277.755} C_VEL
LIN {X 0,Y 297.439,Z 540.706,A -85,B 0,C 180,E1 -16279.793,E2 -16279.793} C_VEL
LIN {X 0,Y 296.901,Z 545.033,A -85,B 0,C 180,E1 -16281.835,E2 -16281.835} C_VEL
LIN {X 0,Y 296.69,Z 547.402,A -85,B 0,C 180,E1 -16283.198,E2 -16283.198} C_VEL
LIN {X 0,Y 296.554,Z 549.203,A -85,B 0,C 180,E1 -16284.561,E2 -16284.561} C_VEL
LIN {X 0,Y 296.528,Z 551.653,A -85,B 0,C 180,E1 -16287.283,E2 -16287.283} C_VEL
LIN {X 0,Y 296.486,Z 552.242,A -85,B 0,C 180,E1 -16288.642,E2 -16288.642} C_VEL
LIN {X 0,Y 296.486,Z 552.242,A -85,B 0,C 180,E1 -16291.358,E2 -16291.358} C_VEL
LIN {X 0,Y 296.528,Z 551.653,A -85,B 0,C 180,E1 -16292.717,E2 -16292.717} C_VEL
LIN {X 0,Y 296.549,Z 549.112,A -85,B 0,C 180,E1 -16295.508,E2 -16295.508} C_VEL
LIN {X 0,Y 296.79,Z 546.251,A -85,B 0,C 180,E1 -16297.483,E2 -16297.483} C_VEL
LIN {X 0,Y 297.255,Z 542.262,A -85,B 0,C 180,E1 -16299.526,E2 -16299.526} C_VEL
LIN {X 0,Y 297.957,Z 537.13,A -85,B 0,C 180,E1 -16301.565,E2 -16301.565} C_VEL
LIN {X 0,Y 298.804,Z 531.868,A -85,B 0,C 180,E1 -16303.257,E2 -16303.257} C_VEL
LIN {X 0,Y 299.922,Z 525.552,A -85,B 0,C 180,E1 -16304.937,E2 -16304.937} C_VEL
LIN {X 0,Y 300.922,Z 519.602,A -85,B 0,C 180,E1 -16306.275,E2 -16306.275} C_VEL
LIN {X 0,Y 301.965,Z 512.672,A -85,B 0,C 180,E1 -16307.611,E2 -16307.611} C_VEL
LIN {X 0,Y 303.291,Z 504.494,A -85,B 0,C 180,E1 -16308.93,E2 -16308.93} C_VEL
LIN {X 0,Y 304.596,Z 495.986,A -85,B 0,C 180,E1 -16310.072,E2 -16310.072} C_VEL
LIN {X 0,Y 305.855,Z 487.273,A -85,B 0,C 180,E1 -16311.04,E2 -16311.04} C_VEL
LIN {X 0,Y 307.048,Z 477.517,A -85,B 0,C 180,E1 -16311.923,E2 -16311.923} C_VEL
LIN {X 0,Y 308.128,Z 467.439,A -85,B 0,C 180,E1 -16312.637,E2 -16312.637} C_VEL
LIN {X 0,Y 308.92,Z 457.928,A -85,B 0,C 180,E1 -16313.15,E2 -16313.15} C_VEL
LIN {X 0,Y 309.604,Z 447.622,A -85,B 0,C 180,E1 -16313.539,E2 -16313.539} C_VEL
LIN {X 0,Y 310.869,Z 396.868,A -85,B 0,C 180,E1 -16314.738,E2 -16314.738} C_VEL
LIN {X 0,Y 311.027,Z 384.995,A -85,B 0,C 180,E1 -16315.021,E2 -16315.021} C_VEL
LIN {X 0,Y 306.753,Z 361.5,A -85,B 0,C 180,E1 -16315.988,E2 -16315.988} C_VEL
LIN {X 0,Y 302.346,Z 341.929,A -85,B 0,C 180,E1 -16316.919,E2 -16316.919} C_VEL
LIN {X 0,Y 302.248,Z 341.089,A -85,B 0,C 180,E1 -16317.057,E2 -16317.057} C_VEL
LIN {X 0,Y 301.408,Z 335.424,A -85,B 0,C 180,E1 -16319.318,E2 -16319.318} C_VEL
LIN {X 0,Y 299.615,Z 326.455,A -85,B 0,C 180,E1 -16323.049,E2 -16323.049} C_VEL
LIN {X 0,Y 298.447,Z 320.81,A -85,B 0,C 180,E1 -16325.558,E2 -16325.558} C_VEL
LIN {X 0,Y 298.348,Z 320.798,A -85,B 0,C 180,E1 -16329.495,E2 -16329.495} C_VEL
LIN {X 0,Y 298.37,Z 320.818,A -85,B 0,C 180,E1 -16333.096,E2 -16333.096} C_VEL
LIN {X 0,Y 298.401,Z 320.813,A -85,B 0,C 180,E1 -16336.92,E2 -16336.92} C_VEL
LIN {X 0,Y 298.396,Z 320.806,A -85,B 0,C 180,E1 -16341.006,E2 -16341.006} C_VEL
LIN {X 0,Y 298.414,Z 320.807,A -85,B 0,C 180,E1 -16343.929,E2 -16343.929} C_VEL
LIN {X 0,Y 298.39,Z 320.81,A -85,B 0,C 180,E1 -16347.983,E2 -16347.983} C_VEL
LIN {X 0,Y 298.444,Z 320.79,A -85,B 0,C 180,E1 -16351.902,E2 -16351.902} C_VEL
LIN {X 0,Y 298.476,Z 320.791,A -85,B 0,C 180,E1 -16354.922,E2 -16354.922} C_VEL
LIN {X 0,Y 298.432,Z 320.794,A -85,B 0,C 180,E1 -16359.313,E2 -16359.313} C_VEL
LIN {X 0,Y 298.529,Z 320.767,A -85,B 0,C 180,E1 -16362.178,E2 -16362.178} C_VEL
LIN {X 0,Y 298.588,Z 320.786,A -85,B 0,C 180,E1 -16364.994,E2 -16364.994} C_VEL
LIN {X 0,Y 298.585,Z 320.761,A -85,B 0,C 180,E1 -16369.146,E2 -16369.146} C_VEL
LIN {X 0,Y 298.734,Z 320.743,A -85,B 0,C 180,E1 -16371.885,E2 -16371.885} C_VEL
LIN {X 0,Y 298.65,Z 320.781,A -85,B 0,C 180,E1 -16374.598,E2 -16374.598} C_VEL
LIN {X 0,Y 298.916,Z 320.724,A -85,B 0,C 180,E1 -16378.652,E2 -16378.652} C_VEL
LIN {X 0,Y 298.916,Z 320.715,A -85,B 0,C 180,E1 -16381.346,E2 -16381.346} C_VEL
LIN {X 0,Y 298.78,Z 320.762,A -85,B 0,C 180,E1 -16386.754,E2 -16386.754} C_VEL
LIN {X 0,Y 298.628,Z 320.748,A -85,B 0,C 180,E1 -16389.481,E2 -16389.481} C_VEL
LIN {X 0,Y 298.544,Z 320.796,A -85,B 0,C 180,E1 -16393.615,E2 -16393.615} C_VEL
LIN {X 0,Y 298.541,Z 320.791,A -85,B 0,C 180,E1 -16396.408,E2 -16396.408} C_VEL
LIN {X 0,Y 298.504,Z 320.771,A -85,B 0,C 180,E1 -16399.654,E2 -16399.654} C_VEL
LIN {X 0,Y 298.45,Z 320.808,A -85,B 0,C 180,E1 -16403.597,E2 -16403.597} C_VEL
LIN {X 0,Y 298.48,Z 320.781,A -85,B 0,C 180,E1 -16406.574,E2 -16406.574} C_VEL
LIN {X 0,Y 298.413,Z 320.809,A -85,B 0,C 180,E1 -16409.641,E2 -16409.641} C_VEL
LIN {X 0,Y 298.389,Z 320.808,A -85,B 0,C 180,E1 -16412.8,E2 -16412.8} C_VEL
LIN {X 0,Y 298.463,Z 320.805,A -85,B 0,C 180,E1 -16416.814,E2 -16416.814} C_VEL
LIN {X 0,Y 298.445,Z 320.795,A -85,B 0,C 180,E1 -16421.25,E2 -16421.25} C_VEL
LIN {X 0,Y 298.41,Z 320.802,A -85,B 0,C 180,E1 -16425.047,E2 -16425.047} C_VEL
LIN {X 0,Y 298.385,Z 320.768,A -85,B 0,C 180,E1 -16428.912,E2 -16428.912} C_VEL
LIN {X 0,Y 298.435,Z 320.814,A -85,B 0,C 180,E1 -16432.246,E2 -16432.246} C_VEL
LIN {X 0,Y 298.402,Z 320.78,A -85,B 0,C 180,E1 -16435.581,E2 -16435.581} C_VEL
LIN {X 0,Y 298.387,Z 320.813,A -85,B 0,C 180,E1 -16438.791,E2 -16438.791} C_VEL
LIN {X 0,Y 298.477,Z 320.971,A -85,B 0,C 180,E1 -16442.325,E2 -16442.325} C_VEL
LIN {X 0,Y 298.787,Z 322.122,A -85,B 0,C 180,E1 -16442.597,E2 -16442.597} C_VEL
LIN {X 0,Y 303.451,Z 330.718,A -85,B 0,C 180,E1 -16443.298,E2 -16443.298} C_VEL
LIN {X 0,Y 310.704,Z 340.937,A -85,B 0,C 180,E1 -16444.321,E2 -16444.321} C_VEL
LIN {X 0,Y 317.5,Z 348.84,A -85,B 0,C 180,E1 -16445.363,E2 -16445.363} C_VEL
LIN {X 0,Y 322.933,Z 354.835,A -85,B 0,C 180,E1 -16446.276,E2 -16446.276} C_VEL
LIN {X 0,Y 328.338,Z 360.689,A -85,B 0,C 180,E1 -16447.281,E2 -16447.281} C_VEL
LIN {X 0,Y 334.819,Z 367.265,A -85,B 0,C 180,E1 -16448.586,E2 -16448.586} C_VEL
LIN {X 0,Y 341.639,Z 373.873,A -85,B 0,C 180,E1 -16450.064,E2 -16450.064} C_VEL
LIN {X 0,Y 348.766,Z 380.369,A -85,B 0,C 180,E1 -16451.752,E2 -16451.752} C_VEL
LIN {X 0,Y 353.428,Z 384.214,A -85,B 0,C 180,E1 -16452.937,E2 -16452.937} C_VEL
LIN {X 0,Y 358.331,Z 388.47,A -85,B 0,C 180,E1 -16454.304,E2 -16454.304} C_VEL
LIN {X 0,Y 362.406,Z 391.595,A -85,B 0,C 180,E1 -16455.537,E2 -16455.537} C_VEL
LIN {X 0,Y 366.987,Z 395.487,A -85,B 0,C 180,E1 -16457.086,E2 -16457.086} C_VEL
LIN {X 0,Y 370.837,Z 398.083,A -85,B 0,C 180,E1 -16458.529,E2 -16458.529} C_VEL
LIN {X 0,Y 373.394,Z 399.789,A -85,B 0,C 180,E1 -16459.599,E2 -16459.599} C_VEL
LIN {X 0,Y 376.665,Z 402.806,A -85,B 0,C 180,E1 -16461.22,E2 -16461.22} C_VEL
LIN {X 0,Y 379.791,Z 404.997,A -85,B 0,C 180,E1 -16463.073,E2 -16463.073} C_VEL
LIN {X 0,Y 382.282,Z 406.333,A -85,B 0,C 180,E1 -16465,E2 -16465} C_VEL
LIN {X 0,Y 383.984,Z 406.855,A -85,B 0,C 180,E1 -16466.852,E2 -16466.852} C_VEL
LIN {X 0,Y 384.932,Z 407.473,A -85,B 0,C 180,E1 -16468.954,E2 -16468.954} C_VEL
LIN {X 0,Y 385.081,Z 407.414,A -85,B 0,C 180,E1 -16470,E2 -16470} C_VEL
LIN {X 0,Y 384.785,Z 407.351,A -85,B 0,C 180,E1 -16471.57,E2 -16471.57} C_VEL
LIN {X 0,Y 383.979,Z 406.888,A -85,B 0,C 180,E1 -16473.148,E2 -16473.148} C_VEL
LIN {X 0,Y 382.281,Z 406.336,A -85,B 0,C 180,E1 -16475,E2 -16475} C_VEL
LIN {X 0,Y 379.792,Z 404.99,A -85,B 0,C 180,E1 -16476.927,E2 -16476.927} C_VEL
LIN {X 0,Y 376.551,Z 402.737,A -85,B 0,C 180,E1 -16478.839,E2 -16478.839} C_VEL
LIN {X 0,Y 372.963,Z 399.383,A -85,B 0,C 180,E1 -16480.595,E2 -16480.595} C_VEL
LIN {X 0,Y 368.236,Z 396.433,A -85,B 0,C 180,E1 -16482.456,E2 -16482.456} C_VEL
LIN {X 0,Y 363.698,Z 392.801,A -85,B 0,C 180,E1 -16484.037,E2 -16484.037} C_VEL
LIN {X 0,Y 360.204,Z 389.823,A -85,B 0,C 180,E1 -16485.144,E2 -16485.144} C_VEL
LIN {X 0,Y 354.989,Z 385.739,A -85,B 0,C 180,E1 -16486.632,E2 -16486.632} C_VEL
LIN {X 0,Y 350.413,Z 381.62,A -85,B 0,C 180,E1 -16487.848,E2 -16487.848} C_VEL
LIN {X 0,Y 344.835,Z 376.8,A -85,B 0,C 180,E1 -16489.203,E2 -16489.203} C_VEL
LIN {X 0,Y 337.919,Z 370.42,A -85,B 0,C 180,E1 -16490.748,E2 -16490.748} C_VEL
LIN {X 0,Y 330.374,Z 362.835,A -85,B 0,C 180,E1 -16492.314,E2 -16492.314} C_VEL
LIN {X 0,Y 323.725,Z 355.801,A -85,B 0,C 180,E1 -16493.574,E2 -16493.574} C_VEL
LIN {X 0,Y 317.62,Z 348.955,A -85,B 0,C 180,E1 -16494.619,E2 -16494.619} C_VEL
LIN {X 0,Y 313.112,Z 343.684,A -85,B 0,C 180,E1 -16495.322,E2 -16495.322} C_VEL
LIN {X 0,Y 308.935,Z 338.533,A -85,B 0,C 180,E1 -16495.936,E2 -16495.936} C_VEL
LIN {X 0,Y 302.852,Z 329.713,A -85,B 0,C 180,E1 -16496.786,E2 -16496.786} C_VEL
LIN {X 0,Y 298.711,Z 321.928,A -85,B 0,C 180,E1 -16497.429,E2 -16497.429} C_VEL
LIN {X 0,Y 298.485,Z 320.903,A -85,B 0,C 180,E1 -16497.727,E2 -16497.727} C_VEL
LIN {X 0,Y 298.389,Z 320.817,A -85,B 0,C 180,E1 -16502.016,E2 -16502.016} C_VEL
LIN {X 0,Y 298.428,Z 320.788,A -85,B 0,C 180,E1 -16506.068,E2 -16506.068} C_VEL
LIN {X 0,Y 298.409,Z 320.797,A -85,B 0,C 180,E1 -16509.485,E2 -16509.485} C_VEL
LIN {X 0,Y 298.42,Z 320.765,A -85,B 0,C 180,E1 -16513.109,E2 -16513.109} C_VEL
LIN {X 0,Y 298.461,Z 320.809,A -85,B 0,C 180,E1 -16516.932,E2 -16516.932} C_VEL
LIN {X 0,Y 298.429,Z 320.806,A -85,B 0,C 180,E1 -16520.998,E2 -16520.998} C_VEL
LIN {X 0,Y 298.427,Z 320.803,A -85,B 0,C 180,E1 -16523.932,E2 -16523.932} C_VEL
LIN {X 0,Y 298.389,Z 320.816,A -85,B 0,C 180,E1 -16527.983,E2 -16527.983} C_VEL
LIN {X 0,Y 298.456,Z 320.784,A -85,B 0,C 180,E1 -16531.904,E2 -16531.904} C_VEL
LIN {X 0,Y 298.478,Z 320.797,A -85,B 0,C 180,E1 -16534.924,E2 -16534.924} C_VEL
LIN {X 0,Y 298.442,Z 320.788,A -85,B 0,C 180,E1 -16539.316,E2 -16539.316} C_VEL
LIN {X 0,Y 298.53,Z 320.776,A -85,B 0,C 180,E1 -16542.18,E2 -16542.18} C_VEL
LIN {X 0,Y 298.586,Z 320.793,A -85,B 0,C 180,E1 -16544.995,E2 -16544.995} C_VEL
LIN {X 0,Y 298.584,Z 320.756,A -85,B 0,C 180,E1 -16549.147,E2 -16549.147} C_VEL
LIN {X 0,Y 298.734,Z 320.754,A -85,B 0,C 180,E1 -16551.886,E2 -16551.886} C_VEL
LIN {X 0,Y 298.65,Z 320.784,A -85,B 0,C 180,E1 -16554.599,E2 -16554.599} C_VEL
LIN {X 0,Y 298.916,Z 320.715,A -85,B 0,C 180,E1 -16558.654,E2 -16558.654} C_VEL
LIN {X 0,Y 298.916,Z 320.724,A -85,B 0,C 180,E1 -16561.348,E2 -16561.348} C_VEL
LIN {X 0,Y 298.781,Z 320.755,A -85,B 0,C 180,E1 -16566.755,E2 -16566.755} C_VEL
LIN {X 0,Y 298.73,Z 320.745,A -85,B 0,C 180,E1 -16567.908,E2 -16567.908} C_VEL
LIN {X 0,Y 298.048,Z 320.825,A -85,B 0,C 180,E1 -16569.032,E2 -16569.032} C_VEL
LIN {X 0,Y 295.094,Z 321.197,A -85,B 0,C 180,E1 -16570.858,E2 -16570.858} C_VEL
LIN {X 0,Y 292.607,Z 321.524,A -85,B 0,C 180,E1 -16572.341,E2 -16572.341} C_VEL
LIN {X 0,Y 291.576,Z 321.661,A -85,B 0,C 180,E1 -16573.492,E2 -16573.492} C_VEL
LIN {X 0,Y 291.512,Z 321.668,A -85,B 0,C 180,E1 -16573.882,E2 -16573.882} C_VEL
LIN {X 0,Y 291.481,Z 321.655,A -85,B 0,C 180,E1 -16576.819,E2 -16576.819} C_VEL
LIN {X 0,Y 291.446,Z 321.655,A -85,B 0,C 180,E1 -16579.876,E2 -16579.876} C_VEL
LIN {X 0,Y 291.377,Z 321.682,A -85,B 0,C 180,E1 -16584.208,E2 -16584.208} C_VEL
LIN {X 0,Y 291.411,Z 321.658,A -85,B 0,C 180,E1 -16587.273,E2 -16587.273} C_VEL
LIN {X 0,Y 291.331,Z 321.698,A -85,B 0,C 180,E1 -16590.438,E2 -16590.438} C_VEL
LIN {X 0,Y 291.341,Z 321.672,A -85,B 0,C 180,E1 -16593.7,E2 -16593.7} C_VEL
LIN {X 0,Y 291.369,Z 321.69,A -85,B 0,C 180,E1 -16597.254,E2 -16597.254} C_VEL
LIN {X 0,Y 291.33,Z 321.684,A -85,B 0,C 180,E1 -16600.644,E2 -16600.644} C_VEL
LIN {X 0,Y 291.289,Z 321.692,A -85,B 0,C 180,E1 -16604.403,E2 -16604.403} C_VEL
LIN {X 0,Y 291.293,Z 321.676,A -85,B 0,C 180,E1 -16608.413,E2 -16608.413} C_VEL
LIN {X 0,Y 291.388,Z 321.679,A -85,B 0,C 180,E1 -16612.918,E2 -16612.918} C_VEL
LIN {X 0,Y 291.424,Z 321.938,A -85,B 0,C 180,E1 -16614.105,E2 -16614.105} C_VEL
LIN {X 0,Y 293.145,Z 329.99,A -85,B 0,C 180,E1 -16617.662,E2 -16617.662} C_VEL
LIN {X 0,Y 294.537,Z 337.157,A -85,B 0,C 180,E1 -16620.716,E2 -16620.716} C_VEL
LIN {X 0,Y 295.232,Z 341.124,A -85,B 0,C 180,E1 -16622.301,E2 -16622.301} C_VEL
LIN {X 0,Y 296.487,Z 345.185,A -85,B 0,C 180,E1 -16622.615,E2 -16622.615} C_VEL
LIN {X 0,Y 301.131,Z 366.576,A -85,B 0,C 180,E1 -16623.626,E2 -16623.626} C_VEL
LIN {X 0,Y 304.674,Z 387.067,A -85,B 0,C 180,E1 -16624.478,E2 -16624.478} C_VEL
LIN {X 0,Y 303.092,Z 447.428,A -85,B 0,C 180,E1 -16625.924,E2 -16625.924} C_VEL
LIN {X 0,Y 302.413,Z 457.734,A -85,B 0,C 180,E1 -16626.322,E2 -16626.322} C_VEL
LIN {X 0,Y 301.579,Z 467.245,A -85,B 0,C 180,E1 -16626.843,E2 -16626.843} C_VEL
LIN {X 0,Y 300.459,Z 477.322,A -85,B 0,C 180,E1 -16627.57,E2 -16627.57} C_VEL
LIN {X 0,Y 299.214,Z 487.078,A -85,B 0,C 180,E1 -16628.47,E2 -16628.47} C_VEL
LIN {X 0,Y 297.905,Z 495.791,A -85,B 0,C 180,E1 -16629.457,E2 -16629.457} C_VEL
LIN {X 0,Y 296.539,Z 504.299,A -85,B 0,C 180,E1 -16630.622,E2 -16630.622} C_VEL
LIN {X 0,Y 295.186,Z 512.478,A -85,B 0,C 180,E1 -16631.971,E2 -16631.971} C_VEL
LIN {X 0,Y 293.802,Z 521.034,A -85,B 0,C 180,E1 -16633.676,E2 -16633.676} C_VEL
LIN {X 0,Y 292.322,Z 529.362,A -85,B 0,C 180,E1 -16635.734,E2 -16635.734} C_VEL
LIN {X 0,Y 291.265,Z 535.018,A -85,B 0,C 180,E1 -16637.458,E2 -16637.458} C_VEL
LIN {X 0,Y 290.436,Z 540.512,A -85,B 0,C 180,E1 -16639.544,E2 -16639.544} C_VEL
LIN {X 0,Y 289.861,Z 544.839,A -85,B 0,C 180,E1 -16641.635,E2 -16641.635} C_VEL
LIN {X 0,Y 289.609,Z 547.207,A -85,B 0,C 180,E1 -16643.031,E2 -16643.031} C_VEL
LIN {X 0,Y 289.457,Z 549.173,A -85,B 0,C 180,E1 -16644.555,E2 -16644.555} C_VEL
LIN {X 0,Y 289.432,Z 551.459,A -85,B 0,C 180,E1 -16647.216,E2 -16647.216} C_VEL
LIN {X 0,Y 289.408,Z 552.049,A -85,B 0,C 180,E1 -16648.609,E2 -16648.609} C_VEL
LIN {X 0,Y 289.408,Z 552.049,A -85,B 0,C 180,E1 -16651.391,E2 -16651.391} C_VEL
LIN {X 0,Y 289.431,Z 551.459,A -85,B 0,C 180,E1 -16652.784,E2 -16652.784} C_VEL
LIN {X 0,Y 289.479,Z 549.009,A -85,B 0,C 180,E1 -16655.573,E2 -16655.573} C_VEL
LIN {X 0,Y 289.721,Z 546.056,A -85,B 0,C 180,E1 -16657.667,E2 -16657.667} C_VEL
LIN {X 0,Y 290.207,Z 542.066,A -85,B 0,C 180,E1 -16659.76,E2 -16659.76} C_VEL
LIN {X 0,Y 290.967,Z 536.935,A -85,B 0,C 180,E1 -16661.847,E2 -16661.847} C_VEL
LIN {X 0,Y 291.881,Z 531.673,A -85,B 0,C 180,E1 -16663.577,E2 -16663.577} C_VEL
LIN {X 0,Y 293.03,Z 525.357,A -85,B 0,C 180,E1 -16665.297,E2 -16665.297} C_VEL
LIN {X 0,Y 294.1,Z 519.407,A -85,B 0,C 180,E1 -16666.664,E2 -16666.664} C_VEL
LIN {X 0,Y 295.182,Z 512.478,A -85,B 0,C 180,E1 -16668.03,E2 -16668.03} C_VEL
LIN {X 0,Y 296.545,Z 504.299,A -85,B 0,C 180,E1 -16669.377,E2 -16669.377} C_VEL
LIN {X 0,Y 297.924,Z 495.791,A -85,B 0,C 180,E1 -16670.542,E2 -16670.542} C_VEL
LIN {X 0,Y 299.212,Z 487.078,A -85,B 0,C 180,E1 -16671.531,E2 -16671.531} C_VEL
LIN {X 0,Y 300.471,Z 477.323,A -85,B 0,C 180,E1 -16672.429,E2 -16672.429} C_VEL
LIN {X 0,Y 301.469,Z 468.533,A -85,B 0,C 180,E1 -16673.075,E2 -16673.075} C_VEL
LIN {X 0,Y 302.342,Z 458.608,A -85,B 0,C 180,E1 -16673.639,E2 -16673.639} C_VEL
LIN {X 0,Y 303.048,Z 448.76,A -85,B 0,C 180,E1 -16674.034,E2 -16674.034} C_VEL
LIN {X 0,Y 303.689,Z 427.733,A -85,B 0,C 180,E1 -16674.571,E2 -16674.571} C_VEL
LIN {X 0,Y 304.576,Z 385.963,A -85,B 0,C 180,E1 -16675.559,E2 -16675.559} C_VEL
LIN {X 0,Y 300.579,Z 363.714,A -85,B 0,C 180,E1 -16676.5,E2 -16676.5} C_VEL
LIN {X 0,Y 296.279,Z 344.522,A -85,B 0,C 180,E1 -16677.423,E2 -16677.423} C_VEL
LIN {X 0,Y 295.252,Z 341.335,A -85,B 0,C 180,E1 -16677.659,E2 -16677.659} C_VEL
LIN {X 0,Y 294.861,Z 339.09,A -85,B 0,C 180,E1 -16678.469,E2 -16678.469} C_VEL
LIN {X 0,Y 293.14,Z 330.006,A -85,B 0,C 180,E1 -16682.332,E2 -16682.332} C_VEL
LIN {X 0,Y 291.391,Z 321.746,A -85,B 0,C 180,E1 -16686.007,E2 -16686.007} C_VEL
LIN {X 0,Y 291.311,Z 321.674,A -85,B 0,C 180,E1 -16689.464,E2 -16689.464} C_VEL
LIN {X 0,Y 291.289,Z 321.703,A -85,B 0,C 180,E1 -16693.628,E2 -16693.628} C_VEL
LIN {X 0,Y 291.319,Z 321.698,A -85,B 0,C 180,E1 -16697.507,E2 -16697.507} C_VEL
LIN {X 0,Y 291.345,Z 321.685,A -85,B 0,C 180,E1 -16701.156,E2 -16701.156} C_VEL
LIN {X 0,Y 291.358,Z 321.68,A -85,B 0,C 180,E1 -16704.625,E2 -16704.625} C_VEL
LIN {X 0,Y 291.367,Z 321.684,A -85,B 0,C 180,E1 -16707.949,E2 -16707.949} C_VEL
LIN {X 0,Y 291.369,Z 321.68,A -85,B 0,C 180,E1 -16711.156,E2 -16711.156} C_VEL
LIN {X 0,Y 291.406,Z 321.663,A -85,B 0,C 180,E1 -16714.27,E2 -16714.27} C_VEL
LIN {X 0,Y 291.369,Z 321.69,A -85,B 0,C 180,E1 -16717.298,E2 -16717.298} C_VEL
LIN {X 0,Y 291.454,Z 321.652,A -85,B 0,C 180,E1 -16720.269,E2 -16720.269} C_VEL
LIN {X 0,Y 291.535,Z 321.663,A -85,B 0,C 180,E1 -16724.633,E2 -16724.633} C_VEL
LIN {X 0,Y 291.529,Z 321.643,A -85,B 0,C 180,E1 -16728.88,E2 -16728.88} C_VEL
LIN {X 0,Y 291.681,Z 321.618,A -85,B 0,C 180,E1 -16731.687,E2 -16731.687} C_VEL
LIN {X 0,Y 291.621,Z 321.656,A -85,B 0,C 180,E1 -16734.467,E2 -16734.467} C_VEL
LIN {X 0,Y 291.883,Z 321.6,A -85,B 0,C 180,E1 -16738.62,E2 -16738.62} C_VEL
LIN {X 0,Y 291.882,Z 321.591,A -85,B 0,C 180,E1 -16741.379,E2 -16741.379} C_VEL
LIN {X 0,Y 291.728,Z 321.638,A -85,B 0,C 180,E1 -16746.918,E2 -16746.918} C_VEL
LIN {X 0,Y 291.567,Z 321.626,A -85,B 0,C 180,E1 -16749.713,E2 -16749.713} C_VEL
LIN {X 0,Y 291.514,Z 321.671,A -85,B 0,C 180,E1 -16753.95,E2 -16753.95} C_VEL
LIN {X 0,Y 291.479,Z 321.664,A -85,B 0,C 180,E1 -16756.817,E2 -16756.817} C_VEL
LIN {X 0,Y 291.444,Z 321.651,A -85,B 0,C 180,E1 -16759.874,E2 -16759.874} C_VEL
LIN {X 0,Y 291.393,Z 321.687,A -85,B 0,C 180,E1 -16764.205,E2 -16764.205} C_VEL
LIN {X 0,Y 291.414,Z 321.657,A -85,B 0,C 180,E1 -16767.271,E2 -16767.271} C_VEL
LIN {X 0,Y 291.331,Z 321.694,A -85,B 0,C 180,E1 -16770.437,E2 -16770.437} C_VEL
LIN {X 0,Y 291.338,Z 321.678,A -85,B 0,C 180,E1 -16773.698,E2 -16773.698} C_VEL
LIN {X 0,Y 291.398,Z 321.689,A -85,B 0,C 180,E1 -16777.261,E2 -16777.261} C_VEL
LIN {X 0,Y 291.394,Z 321.671,A -85,B 0,C 180,E1 -16780.631,E2 -16780.631} C_VEL
LIN {X 0,Y 291.347,Z 321.688,A -85,B 0,C 180,E1 -16784.39,E2 -16784.39} C_VEL
LIN {X 0,Y 291.327,Z 321.642,A -85,B 0,C 180,E1 -16788.403,E2 -16788.403} C_VEL
LIN {X 0,Y 291.368,Z 321.685,A -85,B 0,C 180,E1 -16791.162,E2 -16791.162} C_VEL
LIN {X 0,Y 291.38,Z 321.656,A -85,B 0,C 180,E1 -16794.63,E2 -16794.63} C_VEL
LIN {X 0,Y 291.366,Z 321.692,A -85,B 0,C 180,E1 -16797.951,E2 -16797.951} C_VEL
LIN {X 0,Y 291.422,Z 321.832,A -85,B 0,C 180,E1 -16801.616,E2 -16801.616} C_VEL
LIN {X 0,Y 291.699,Z 322.907,A -85,B 0,C 180,E1 -16801.89,E2 -16801.89} C_VEL
LIN {X 0,Y 297.799,Z 334.351,A -85,B 0,C 180,E1 -16802.841,E2 -16802.841} C_VEL
LIN {X 0,Y 305.438,Z 345.198,A -85,B 0,C 180,E1 -16803.877,E2 -16803.877} C_VEL
LIN {X 0,Y 312.921,Z 353.783,A -85,B 0,C 180,E1 -16804.931,E2 -16804.931} C_VEL
LIN {X 0,Y 320.442,Z 361.999,A -85,B 0,C 180,E1 -16806.128,E2 -16806.128} C_VEL
LIN {X 0,Y 325.527,Z 367.116,A -85,B 0,C 180,E1 -16807.033,E2 -16807.033} C_VEL
LIN {X 0,Y 331.289,Z 372.923,A -85,B 0,C 180,E1 -16808.141,E2 -16808.141} C_VEL
LIN {X 0,Y 338.975,Z 380.175,A -85,B 0,C 180,E1 -16809.745,E2 -16809.745} C_VEL
LIN {X 0,Y 346.402,Z 386.817,A -85,B 0,C 180,E1 -16811.455,E2 -16811.455} C_VEL
LIN {X 0,Y 350.978,Z 390.496,A -85,B 0,C 180,E1 -16812.589,E2 -16812.589} C_VEL
LIN {X 0,Y 356.027,Z 394.83,A -85,B 0,C 180,E1 -16813.957,E2 -16813.957} C_VEL
LIN {X 0,Y 360.679,Z 398.378,A -85,B 0,C 180,E1 -16815.327,E2 -16815.327} C_VEL
LIN {X 0,Y 365.331,Z 402.218,A -85,B 0,C 180,E1 -16816.846,E2 -16816.846} C_VEL
LIN {X 0,Y 369.816,Z 405.125,A -85,B 0,C 180,E1 -16818.497,E2 -16818.497} C_VEL
LIN {X 0,Y 372.05,Z 406.673,A -85,B 0,C 180,E1 -16819.424,E2 -16819.424} C_VEL
LIN {X 0,Y 375.42,Z 409.703,A -85,B 0,C 180,E1 -16821.048,E2 -16821.048} C_VEL
LIN {X 0,Y 378.557,Z 411.879,A -85,B 0,C 180,E1 -16822.854,E2 -16822.854} C_VEL
LIN {X 0,Y 381.111,Z 413.226,A -85,B 0,C 180,E1 -16824.742,E2 -16824.742} C_VEL
LIN {X 0,Y 382.221,Z 413.697,A -85,B 0,C 180,E1 -16825.782,E2 -16825.782} C_VEL
LIN {X 0,Y 383.426,Z 414.101,A -85,B 0,C 180,E1 -16827.361,E2 -16827.361} C_VEL
LIN {X 0,Y 384.07,Z 414.52,A -85,B 0,C 180,E1 -16828.952,E2 -16828.952} C_VEL
LIN {X 0,Y 384.216,Z 414.461,A -85,B 0,C 180,E1 -16830,E2 -16830} C_VEL
LIN {X 0,Y 383.918,Z 414.383,A -85,B 0,C 180,E1 -16831.573,E2 -16831.573} C_VEL
LIN {X 0,Y 383.105,Z 413.909,A -85,B 0,C 180,E1 -16833.155,E2 -16833.155} C_VEL
LIN {X 0,Y 381.391,Z 413.382,A -85,B 0,C 180,E1 -16835.012,E2 -16835.012} C_VEL
LIN {X 0,Y 378.869,Z 412.047,A -85,B 0,C 180,E1 -16836.944,E2 -16836.944} C_VEL
LIN {X 0,Y 375.589,Z 409.83,A -85,B 0,C 180,E1 -16838.862,E2 -16838.862} C_VEL
LIN {X 0,Y 372.101,Z 406.746,A -85,B 0,C 180,E1 -16840.552,E2 -16840.552} C_VEL
LIN {X 0,Y 369.817,Z 405.12,A -85,B 0,C 180,E1 -16841.503,E2 -16841.503} C_VEL
LIN {X 0,Y 365.328,Z 402.239,A -85,B 0,C 180,E1 -16843.155,E2 -16843.155} C_VEL
LIN {X 0,Y 360.24,Z 397.988,A -85,B 0,C 180,E1 -16844.811,E2 -16844.811} C_VEL
LIN {X 0,Y 353.899,Z 393.165,A -85,B 0,C 180,E1 -16846.631,E2 -16846.631} C_VEL
LIN {X 0,Y 348.072,Z 388.074,A -85,B 0,C 180,E1 -16848.143,E2 -16848.143} C_VEL
LIN {X 0,Y 342.747,Z 383.606,A -85,B 0,C 180,E1 -16849.402,E2 -16849.402} C_VEL
LIN {X 0,Y 335.126,Z 376.709,A -85,B 0,C 180,E1 -16851.067,E2 -16851.067} C_VEL
LIN {X 0,Y 330.036,Z 371.782,A -85,B 0,C 180,E1 -16852.105,E2 -16852.105} C_VEL
LIN {X 0,Y 321.069,Z 362.693,A -85,B 0,C 180,E1 -16853.763,E2 -16853.763} C_VEL
LIN {X 0,Y 313.827,Z 354.714,A -85,B 0,C 180,E1 -16854.941,E2 -16854.941} C_VEL
LIN {X 0,Y 308.734,Z 348.959,A -85,B 0,C 180,E1 -16855.679,E2 -16855.679} C_VEL
LIN {X 0,Y 303.975,Z 343.199,A -85,B 0,C 180,E1 -16856.324,E2 -16856.324} C_VEL
LIN {X 0,Y 297.451,Z 333.754,A -85,B 0,C 180,E1 -16857.209,E2 -16857.209} C_VEL
LIN {X 0,Y 291.624,Z 322.697,A -85,B 0,C 180,E1 -16858.143,E2 -16858.143} C_VEL
LIN {X 0,Y 291.405,Z 321.752,A -85,B 0,C 180,E1 -16858.45,E2 -16858.45} C_VEL
LIN {X 0,Y 291.337,Z 321.687,A -85,B 0,C 180,E1 -16862.403,E2 -16862.403} C_VEL
LIN {X 0,Y 291.38,Z 321.656,A -85,B 0,C 180,E1 -16865.37,E2 -16865.37} C_VEL
LIN {X 0,Y 291.368,Z 321.685,A -85,B 0,C 180,E1 -16868.838,E2 -16868.838} C_VEL
LIN {X 0,Y 291.334,Z 321.641,A -85,B 0,C 180,E1 -16872.489,E2 -16872.489} C_VEL
LIN {X 0,Y 291.364,Z 321.691,A -85,B 0,C 180,E1 -16876.353,E2 -16876.353} C_VEL
LIN {X 0,Y 291.4,Z 321.679,A -85,B 0,C 180,E1 -16880.512,E2 -16880.512} C_VEL
LIN {X 0,Y 291.426,Z 321.684,A -85,B 0,C 180,E1 -16882.923,E2 -16882.923} C_VEL
LIN {X 0,Y 291.338,Z 321.678,A -85,B 0,C 180,E1 -16886.302,E2 -16886.302} C_VEL
LIN {X 0,Y 291.38,Z 321.686,A -85,B 0,C 180,E1 -16890.26,E2 -16890.26} C_VEL
LIN {X 0,Y 291.407,Z 321.673,A -85,B 0,C 180,E1 -16894.272,E2 -16894.272} C_VEL
LIN {X 0,Y 291.374,Z 321.688,A -85,B 0,C 180,E1 -16897.3,E2 -16897.3} C_VEL
LIN {X 0,Y 291.451,Z 321.649,A -85,B 0,C 180,E1 -16900.271,E2 -16900.271} C_VEL
LIN {X 0,Y 291.533,Z 321.668,A -85,B 0,C 180,E1 -16904.635,E2 -16904.635} C_VEL
LIN {X 0,Y 291.528,Z 321.637,A -85,B 0,C 180,E1 -16908.881,E2 -16908.881} C_VEL
LIN {X 0,Y 291.68,Z 321.627,A -85,B 0,C 180,E1 -16911.688,E2 -16911.688} C_VEL
LIN {X 0,Y 291.62,Z 321.659,A -85,B 0,C 180,E1 -16914.469,E2 -16914.469} C_VEL
LIN {X 0,Y 291.882,Z 321.591,A -85,B 0,C 180,E1 -16918.621,E2 -16918.621} C_VEL
LIN {X 0,Y 291.883,Z 321.6,A -85,B 0,C 180,E1 -16921.38,E2 -16921.38} C_VEL
LIN {X 0,Y 291.729,Z 321.631,A -85,B 0,C 180,E1 -16926.919,E2 -16926.919} C_VEL
LIN {X 0,Y 291.569,Z 321.625,A -85,B 0,C 180,E1 -16929.715,E2 -16929.715} C_VEL
LIN {X 0,Y 291.512,Z 321.668,A -85,B 0,C 180,E1 -16933.882,E2 -16933.882} C_VEL
LIN {X 0,Y 290.877,Z 321.752,A -85,B 0,C 180,E1 -16935.035,E2 -16935.035} C_VEL
LIN {X 0,Y 287.966,Z 322.098,A -85,B 0,C 180,E1 -16936.909,E2 -16936.909} C_VEL
LIN {X 0,Y 285.486,Z 322.392,A -85,B 0,C 180,E1 -16938.431,E2 -16938.431} C_VEL
LIN {X 0,Y 284.447,Z 322.523,A -85,B 0,C 180,E1 -16939.613,E2 -16939.613} C_VEL
LIN {X 0,Y 284.379,Z 322.536,A -85,B 0,C 180,E1 -16940.013,E2 -16940.013} C_VEL
LIN {X 0,Y 284.33,Z 322.565,A -85,B 0,C 180,E1 -16943.86,E2 -16943.86} C_VEL
LIN {X 0,Y 284.388,Z 322.531,A -85,B 0,C 180,E1 -16947.173,E2 -16947.173} C_VEL
LIN {X 0,Y 284.29,Z 322.571,A -85,B 0,C 180,E1 -16951.276,E2 -16951.276} C_VEL
LIN {X 0,Y 284.338,Z 322.553,A -85,B 0,C 180,E1 -16955.349,E2 -16955.349} C_VEL
LIN {X 0,Y 284.305,Z 322.567,A -85,B 0,C 180,E1 -16958.171,E2 -16958.171} C_VEL
LIN {X 0,Y 284.268,Z 322.576,A -85,B 0,C 180,E1 -16962.126,E2 -16962.126} C_VEL
LIN {X 0,Y 284.237,Z 322.582,A -85,B 0,C 180,E1 -16966.187,E2 -16966.187} C_VEL
LIN {X 0,Y 284.255,Z 322.548,A -85,B 0,C 180,E1 -16970.037,E2 -16970.037} C_VEL
LIN {X 0,Y 284.375,Z 322.745,A -85,B 0,C 180,E1 -16973.511,E2 -16973.511} C_VEL
LIN {X 0,Y 286.128,Z 331.013,A -85,B 0,C 180,E1 -16977.292,E2 -16977.292} C_VEL
LIN {X 0,Y 287.638,Z 338.873,A -85,B 0,C 180,E1 -16980.748,E2 -16980.748} C_VEL
LIN {X 0,Y 288.064,Z 341.153,A -85,B 0,C 180,E1 -16981.593,E2 -16981.593} C_VEL
LIN {X 0,Y 290.561,Z 348.007,A -85,B 0,C 180,E1 -16982.09,E2 -16982.09} C_VEL
LIN {X 0,Y 295.581,Z 371.787,A -85,B 0,C 180,E1 -16983.235,E2 -16983.235} C_VEL
LIN {X 0,Y 298.239,Z 387.526,A -85,B 0,C 180,E1 -16983.904,E2 -16983.904} C_VEL
LIN {X 0,Y 296.639,Z 447.234,A -85,B 0,C 180,E1 -16985.366,E2 -16985.366} C_VEL
LIN {X 0,Y 295.935,Z 457.54,A -85,B 0,C 180,E1 -16985.771,E2 -16985.771} C_VEL
LIN {X 0,Y 295.069,Z 467.051,A -85,B 0,C 180,E1 -16986.302,E2 -16986.302} C_VEL
LIN {X 0,Y 293.887,Z 477.128,A -85,B 0,C 180,E1 -16987.04,E2 -16987.04} C_VEL
LIN {X 0,Y 292.622,Z 486.884,A -85,B 0,C 180,E1 -16987.959,E2 -16987.959} C_VEL
LIN {X 0,Y 291.055,Z 496.948,A -85,B 0,C 180,E1 -16989.136,E2 -16989.136} C_VEL
LIN {X 0,Y 289.078,Z 508.444,A -85,B 0,C 180,E1 -16990.84,E2 -16990.84} C_VEL
LIN {X 0,Y 287.687,Z 516.386,A -85,B 0,C 180,E1 -16992.318,E2 -16992.318} C_VEL
LIN {X 0,Y 286.375,Z 523.785,A -85,B 0,C 180,E1 -16993.974,E2 -16993.974} C_VEL
LIN {X 0,Y 285.181,Z 530.323,A -85,B 0,C 180,E1 -16995.733,E2 -16995.733} C_VEL
LIN {X 0,Y 284.301,Z 534.823,A -85,B 0,C 180,E1 -16997.145,E2 -16997.145} C_VEL
LIN {X 0,Y 283.424,Z 540.317,A -85,B 0,C 180,E1 -16999.282,E2 -16999.282} C_VEL
LIN {X 0,Y 282.81,Z 544.644,A -85,B 0,C 180,E1 -17001.425,E2 -17001.425} C_VEL
LIN {X 0,Y 282.557,Z 547.013,A -85,B 0,C 180,E1 -17002.856,E2 -17002.856} C_VEL
LIN {X 0,Y 282.362,Z 549.244,A -85,B 0,C 180,E1 -17004.631,E2 -17004.631} C_VEL
LIN {X 0,Y 282.338,Z 551.265,A -85,B 0,C 180,E1 -17007.146,E2 -17007.146} C_VEL
